HMI tags "2925RS001A01L02"
   "2925RS001A01L02.MSW" : 52809b66-421d-457f-8884-6f7a49d4e247 AT %DB5066.DBX18.0, 500 ms
   "2925RS001A01L02.DefaultText" : TextRef, internal   // Заголовок POPUP окна. При експорте из ECS через скрипт заполняется автоматически, если теги копируются в ручную то требуется в ручную задатать свойство Start Value
   "2925RS001A01L02.BlockInfo" : Array [0..2] of Int AT %DB5066.DBX38.0, 500 ms
   "2925RS001A01L02.StatusWork" : Int AT %DB5066.DBW242, 500 ms
   "2925RS001A01L02.FP_PARAM.DampingTime" : Int AT %DB5066.DBW50, 500 ms
   "2925RS001A01L02.FP_PARAM.Force_Value" : Real AT %DB5066.DBD52, 500 ms
   "2925RS001A01L02.FP_PARAM.Scale_Min" : Real AT %DB5066.DBD56, 500 ms
   "2925RS001A01L02.FP_PARAM.Scale_Max" : Real AT %DB5066.DBD60, 500 ms
   "2925RS001A01L02.FP_PARAM.Gradient" : Real AT %DB5066.DBD64, 500 ms
   "2925RS001A01L02.FP_PARAM.Grad_Pos" : Real AT %DB5066.DBD68, 500 ms
   "2925RS001A01L02.FP_PARAM.Grad_Neg" : Real AT %DB5066.DBD72, 500 ms
   "2925RS001A01L02.FP_PARAM.Grad_X" : Real AT %DB5066.DBD76, 500 ms
   "2925RS001A01L02.FP_PARAM.Gradient_Time_Pre" : Int AT %DB5066.DBW80, 500 ms
   "2925RS001A01L02.FP_PARAM.Gradient_Time_ACC" : Int AT %DB5066.DBW82, 500 ms
   "2925RS001A01L02.FP_PARAM.Alarm_Hyst" : Real AT %DB5066.DBD84, 500 ms
   "2925RS001A01L02.FP_PARAM.AlarmLimit_H3" : Real AT %DB5066.DBD88, 500 ms
   "2925RS001A01L02.FP_PARAM.AlarmLimit_H2" : Real AT %DB5066.DBD92, 500 ms
   "2925RS001A01L02.FP_PARAM.AlarmLimit_H1" : Real AT %DB5066.DBD96, 500 ms
   "2925RS001A01L02.FP_PARAM.AlarmLimit_L1" : Real AT %DB5066.DBD100, 500 ms
   "2925RS001A01L02.FP_PARAM.AlarmLimit_L2" : Real AT %DB5066.DBD104, 500 ms
   "2925RS001A01L02.FP_PARAM.AlarmLimit_L3" : Real AT %DB5066.DBD108, 500 ms
   "2925RS001A01L02.FP_PARAM.AlarmDelay_H3_Pre" : Int AT %DB5066.DBW112, 500 ms
   "2925RS001A01L02.FP_PARAM.AlarmDelay_H3_Acc" : Int AT %DB5066.DBW114, 500 ms
   "2925RS001A01L02.FP_PARAM.AlarmDelay_H2_Pre" : Int AT %DB5066.DBW116, 500 ms
   "2925RS001A01L02.FP_PARAM.AlarmDelay_H2_Acc" : Int AT %DB5066.DBW118, 500 ms
   "2925RS001A01L02.FP_PARAM.AlarmDelay_H1_Pre" : Int AT %DB5066.DBW120, 500 ms
   "2925RS001A01L02.FP_PARAM.AlarmDelay_H1_Acc" : Int AT %DB5066.DBW122, 500 ms
   "2925RS001A01L02.FP_PARAM.AlarmDelay_L1_Pre" : Int AT %DB5066.DBW124, 500 ms
   "2925RS001A01L02.FP_PARAM.AlarmDelay_L1_Acc" : Int AT %DB5066.DBW126, 500 ms
   "2925RS001A01L02.FP_PARAM.AlarmDelay_L2_Pre" : Int AT %DB5066.DBW128, 500 ms
   "2925RS001A01L02.FP_PARAM.AlarmDelay_L2_Acc" : Int AT %DB5066.DBW130, 500 ms
   "2925RS001A01L02.FP_PARAM.AlarmDelay_L3_Pre" : Int AT %DB5066.DBW132, 500 ms
   "2925RS001A01L02.FP_PARAM.AlarmDelay_L3_Acc" : Int AT %DB5066.DBW134, 500 ms
   "2925RS001A01L02.FP_PARAM.OpenLoopDelay_Pre" : Int AT %DB5066.DBW136, 500 ms
   "2925RS001A01L02.FP_PARAM.OpenLoopDelay_Acc" : Int AT %DB5066.DBW138, 500 ms
   "2925RS001A01L02.FP_PARAM.OverRangeDelay_Pre" : Int AT %DB5066.DBW140, 500 ms
   "2925RS001A01L02.FP_PARAM.OverRangeDelay_Acc" : Int AT %DB5066.DBW142, 500 ms
   "2925RS001A01L02.FP_PARAM.AuxLimit_H2_Value" : Real AT %DB5066.DBD144, 500 ms
   "2925RS001A01L02.FP_PARAM.AuxLimit_H1_Value" : Real AT %DB5066.DBD148, 500 ms
   "2925RS001A01L02.FP_PARAM.AuxLimit_L2_Value" : Real AT %DB5066.DBD152, 500 ms
   "2925RS001A01L02.FP_PARAM.AuxLimit_L1_Value" : Real AT %DB5066.DBD156, 500 ms
   "2925RS001A01L02.Unit" : TextRef, internal   // Еденицы измерения При експорте из ECS через скрипт заполняется автоматически, если теги копируются в ручную то требуется задатать свойство Text
   "2925RS001A01L02.Decimals" : TextRef, internal   // Формат отображения При експорте из ECS через скрипт, заполняется автоматически. Если теги копируются в ручную то требуется задатать свойство Text s999999.9
   "2925RS001A01L02.FP_EN.Square" : Bool AT %DB5066.DBX46.0, 500 ms
   "2925RS001A01L02.FP_EN.SquareRoot" : Bool AT %DB5066.DBX46.1, 500 ms
   "2925RS001A01L02.FP_EN.ParentSupress" : Bool AT %DB5066.DBX46.2, 500 ms
   "2925RS001A01L02.FP_EN.ParentSupressUnit" : Bool AT %DB5066.DBX46.3, 500 ms
   "2925RS001A01L02.FP_EN.Force" : Bool AT %DB5066.DBX46.4, 500 ms
   "2925RS001A01L02.FP_EN.Damping" : Bool AT %DB5066.DBX46.5, 500 ms
   "2925RS001A01L02.FP_EN.Gradient_Pos" : Bool AT %DB5066.DBX46.6, 500 ms
   "2925RS001A01L02.FP_EN.Gradient_Neg" : Bool AT %DB5066.DBX46.7, 500 ms
   "2925RS001A01L02.FP_EN.Hysteresis" : Bool AT %DB5066.DBX47.0, 500 ms
   "2925RS001A01L02.FP_EN.Alarm_H3" : Bool AT %DB5066.DBX47.1, 500 ms
   "2925RS001A01L02.FP_EN.Alarm_H2" : Bool AT %DB5066.DBX47.2, 500 ms
   "2925RS001A01L02.FP_EN.Alarm_H1" : Bool AT %DB5066.DBX47.3, 500 ms
   "2925RS001A01L02.FP_EN.Alarm_L1" : Bool AT %DB5066.DBX47.4, 500 ms
   "2925RS001A01L02.FP_EN.Alarm_L2" : Bool AT %DB5066.DBX47.5, 500 ms
   "2925RS001A01L02.FP_EN.Alarm_L3" : Bool AT %DB5066.DBX47.6, 500 ms
   "2925RS001A01L02.FP_EN.AlarmDelay_H3" : Bool AT %DB5066.DBX47.7, 500 ms
   "2925RS001A01L02.FP_EN.AlarmDelay_H2" : Bool AT %DB5066.DBX48.0, 500 ms
   "2925RS001A01L02.FP_EN.AlarmDelay_H1" : Bool AT %DB5066.DBX48.1, 500 ms
   "2925RS001A01L02.FP_EN.AlarmDelay_L1" : Bool AT %DB5066.DBX48.2, 500 ms
   "2925RS001A01L02.FP_EN.AlarmDelay_L2" : Bool AT %DB5066.DBX48.3, 500 ms
   "2925RS001A01L02.FP_EN.AlarmDelay_L3" : Bool AT %DB5066.DBX48.4, 500 ms
   "2925RS001A01L02.FP_EN.ROC_Warn" : Bool AT %DB5066.DBX48.5, 500 ms
   "2925RS001A01L02.FP_EN.U_Range_Warn" : Bool AT %DB5066.DBX48.6, 500 ms
   "2925RS001A01L02.FP_EN.O_Range_Warn" : Bool AT %DB5066.DBX48.7, 500 ms
   "2925RS001A01L02.trend_tag_name" : TextRef, internal   // Еденицы измерения При експорте из ECS через скрипт - заполняется автоматически, если теги копируются в ручную то требуется задатать свойство Text - имя тега для тренда
   "2925RS001A01L02.DQ.AL_H3" : Bool AT %DB5066.DBX16.0, 500 ms
   "2925RS001A01L02.DQ.AL_H2" : Bool AT %DB5066.DBX16.1, 500 ms
   "2925RS001A01L02.DQ.AL_H1" : Bool AT %DB5066.DBX16.2, 500 ms
   "2925RS001A01L02.DQ.AL_L1" : Bool AT %DB5066.DBX16.3, 500 ms
   "2925RS001A01L02.DQ.AL_L2" : Bool AT %DB5066.DBX16.4, 500 ms
   "2925RS001A01L02.DQ.AL_L3" : Bool AT %DB5066.DBX16.5, 500 ms
   "2925RS001A01L02.DQ.SIG_OK" : Bool AT %DB5066.DBX16.6, 500 ms
   "2925RS001A01L02.DQ.LIM_H2" : Bool AT %DB5066.DBX16.7, 500 ms
   "2925RS001A01L02.DQ.LIM_H1" : Bool AT %DB5066.DBX17.0, 500 ms
   "2925RS001A01L02.DQ.LIM_L1" : Bool AT %DB5066.DBX17.1, 500 ms
   "2925RS001A01L02.DQ.LIM_L2" : Bool AT %DB5066.DBX17.2, 500 ms
   "2925RS001A01L02.DQ.GR_P" : Bool AT %DB5066.DBX17.3, 500 ms
   "2925RS001A01L02.DQ.GR_N" : Bool AT %DB5066.DBX17.4, 500 ms
   "2925RS001A01L02.I.IN" : Real AT %DB5066.DBD2, 500 ms
   "2925RS001A01L02.I.SIG_TYPE" : Int AT %DB5066.DBW0, 500 ms
   "2925RS001A01L02.I.FI_BUS" : Byte AT %DB5066.DBB6, 500 ms
   "2925RS001A01L02.DI.U_RANGE" : Bool AT %DB5066.DBX7.0, 500 ms
   "2925RS001A01L02.DI.O_RANGE" : Bool AT %DB5066.DBX7.1, 500 ms
   "2925RS001A01L02.DI.SIG_FAULT" : Bool AT %DB5066.DBX7.2, 500 ms
   "2925RS001A01L02.DI.EnConfig" : Bool AT %DB5066.DBX7.3, 500 ms
   "2925RS001A01L02.DI.AEN" : Bool AT %DB5066.DBX7.4, 500 ms
   "2925RS001A01L02.DI.AL_SUPR" : Bool AT %DB5066.DBX7.5, 500 ms
   "2925RS001A01L02.Q.PV_NORM" : Real AT %DB5066.DBD8, 500 ms
   "2925RS001A01L02.Q.PV_SCAL" : Real AT %DB5066.DBD12, 500 ms
   "2925RS001A01L02.ParentInfo" : TextRef, internal   // Имя родителя для попап окна, вкладка инфо. При експорте из ECS через скрипт заполняется автоматически, если теги копируются в ручную то требуется в ручную задатать свойство Start Value

HMI tags "2925RS001A01T01"
   "2925RS001A01T01.MSW" : 52809b66-421d-457f-8884-6f7a49d4e247 AT %DB5067.DBX18.0, 500 ms
   "2925RS001A01T01.DefaultText" : TextRef, internal   // Заголовок POPUP окна. При експорте из ECS через скрипт заполняется автоматически, если теги копируются в ручную то требуется в ручную задатать свойство Start Value
   "2925RS001A01T01.BlockInfo" : Array [0..2] of Int AT %DB5067.DBX38.0, 500 ms
   "2925RS001A01T01.StatusWork" : Int AT %DB5067.DBW242, 500 ms
   "2925RS001A01T01.FP_PARAM.DampingTime" : Int AT %DB5067.DBW50, 500 ms
   "2925RS001A01T01.FP_PARAM.Force_Value" : Real AT %DB5067.DBD52, 500 ms
   "2925RS001A01T01.FP_PARAM.Scale_Min" : Real AT %DB5067.DBD56, 500 ms
   "2925RS001A01T01.FP_PARAM.Scale_Max" : Real AT %DB5067.DBD60, 500 ms
   "2925RS001A01T01.FP_PARAM.Gradient" : Real AT %DB5067.DBD64, 500 ms
   "2925RS001A01T01.FP_PARAM.Grad_Pos" : Real AT %DB5067.DBD68, 500 ms
   "2925RS001A01T01.FP_PARAM.Grad_Neg" : Real AT %DB5067.DBD72, 500 ms
   "2925RS001A01T01.FP_PARAM.Grad_X" : Real AT %DB5067.DBD76, 500 ms
   "2925RS001A01T01.FP_PARAM.Gradient_Time_Pre" : Int AT %DB5067.DBW80, 500 ms
   "2925RS001A01T01.FP_PARAM.Gradient_Time_ACC" : Int AT %DB5067.DBW82, 500 ms
   "2925RS001A01T01.FP_PARAM.Alarm_Hyst" : Real AT %DB5067.DBD84, 500 ms
   "2925RS001A01T01.FP_PARAM.AlarmLimit_H3" : Real AT %DB5067.DBD88, 500 ms
   "2925RS001A01T01.FP_PARAM.AlarmLimit_H2" : Real AT %DB5067.DBD92, 500 ms
   "2925RS001A01T01.FP_PARAM.AlarmLimit_H1" : Real AT %DB5067.DBD96, 500 ms
   "2925RS001A01T01.FP_PARAM.AlarmLimit_L1" : Real AT %DB5067.DBD100, 500 ms
   "2925RS001A01T01.FP_PARAM.AlarmLimit_L2" : Real AT %DB5067.DBD104, 500 ms
   "2925RS001A01T01.FP_PARAM.AlarmLimit_L3" : Real AT %DB5067.DBD108, 500 ms
   "2925RS001A01T01.FP_PARAM.AlarmDelay_H3_Pre" : Int AT %DB5067.DBW112, 500 ms
   "2925RS001A01T01.FP_PARAM.AlarmDelay_H3_Acc" : Int AT %DB5067.DBW114, 500 ms
   "2925RS001A01T01.FP_PARAM.AlarmDelay_H2_Pre" : Int AT %DB5067.DBW116, 500 ms
   "2925RS001A01T01.FP_PARAM.AlarmDelay_H2_Acc" : Int AT %DB5067.DBW118, 500 ms
   "2925RS001A01T01.FP_PARAM.AlarmDelay_H1_Pre" : Int AT %DB5067.DBW120, 500 ms
   "2925RS001A01T01.FP_PARAM.AlarmDelay_H1_Acc" : Int AT %DB5067.DBW122, 500 ms
   "2925RS001A01T01.FP_PARAM.AlarmDelay_L1_Pre" : Int AT %DB5067.DBW124, 500 ms
   "2925RS001A01T01.FP_PARAM.AlarmDelay_L1_Acc" : Int AT %DB5067.DBW126, 500 ms
   "2925RS001A01T01.FP_PARAM.AlarmDelay_L2_Pre" : Int AT %DB5067.DBW128, 500 ms
   "2925RS001A01T01.FP_PARAM.AlarmDelay_L2_Acc" : Int AT %DB5067.DBW130, 500 ms
   "2925RS001A01T01.FP_PARAM.AlarmDelay_L3_Pre" : Int AT %DB5067.DBW132, 500 ms
   "2925RS001A01T01.FP_PARAM.AlarmDelay_L3_Acc" : Int AT %DB5067.DBW134, 500 ms
   "2925RS001A01T01.FP_PARAM.OpenLoopDelay_Pre" : Int AT %DB5067.DBW136, 500 ms
   "2925RS001A01T01.FP_PARAM.OpenLoopDelay_Acc" : Int AT %DB5067.DBW138, 500 ms
   "2925RS001A01T01.FP_PARAM.OverRangeDelay_Pre" : Int AT %DB5067.DBW140, 500 ms
   "2925RS001A01T01.FP_PARAM.OverRangeDelay_Acc" : Int AT %DB5067.DBW142, 500 ms
   "2925RS001A01T01.FP_PARAM.AuxLimit_H2_Value" : Real AT %DB5067.DBD144, 500 ms
   "2925RS001A01T01.FP_PARAM.AuxLimit_H1_Value" : Real AT %DB5067.DBD148, 500 ms
   "2925RS001A01T01.FP_PARAM.AuxLimit_L2_Value" : Real AT %DB5067.DBD152, 500 ms
   "2925RS001A01T01.FP_PARAM.AuxLimit_L1_Value" : Real AT %DB5067.DBD156, 500 ms
   "2925RS001A01T01.Unit" : TextRef, internal   // Еденицы измерения При експорте из ECS через скрипт заполняется автоматически, если теги копируются в ручную то требуется задатать свойство Text
   "2925RS001A01T01.Decimals" : TextRef, internal   // Формат отображения При експорте из ECS через скрипт, заполняется автоматически. Если теги копируются в ручную то требуется задатать свойство Text s999999.9
   "2925RS001A01T01.FP_EN.Square" : Bool AT %DB5067.DBX46.0, 500 ms
   "2925RS001A01T01.FP_EN.SquareRoot" : Bool AT %DB5067.DBX46.1, 500 ms
   "2925RS001A01T01.FP_EN.ParentSupress" : Bool AT %DB5067.DBX46.2, 500 ms
   "2925RS001A01T01.FP_EN.ParentSupressUnit" : Bool AT %DB5067.DBX46.3, 500 ms
   "2925RS001A01T01.FP_EN.Force" : Bool AT %DB5067.DBX46.4, 500 ms
   "2925RS001A01T01.FP_EN.Damping" : Bool AT %DB5067.DBX46.5, 500 ms
   "2925RS001A01T01.FP_EN.Gradient_Pos" : Bool AT %DB5067.DBX46.6, 500 ms
   "2925RS001A01T01.FP_EN.Gradient_Neg" : Bool AT %DB5067.DBX46.7, 500 ms
   "2925RS001A01T01.FP_EN.Hysteresis" : Bool AT %DB5067.DBX47.0, 500 ms
   "2925RS001A01T01.FP_EN.Alarm_H3" : Bool AT %DB5067.DBX47.1, 500 ms
   "2925RS001A01T01.FP_EN.Alarm_H2" : Bool AT %DB5067.DBX47.2, 500 ms
   "2925RS001A01T01.FP_EN.Alarm_H1" : Bool AT %DB5067.DBX47.3, 500 ms
   "2925RS001A01T01.FP_EN.Alarm_L1" : Bool AT %DB5067.DBX47.4, 500 ms
   "2925RS001A01T01.FP_EN.Alarm_L2" : Bool AT %DB5067.DBX47.5, 500 ms
   "2925RS001A01T01.FP_EN.Alarm_L3" : Bool AT %DB5067.DBX47.6, 500 ms
   "2925RS001A01T01.FP_EN.AlarmDelay_H3" : Bool AT %DB5067.DBX47.7, 500 ms
   "2925RS001A01T01.FP_EN.AlarmDelay_H2" : Bool AT %DB5067.DBX48.0, 500 ms
   "2925RS001A01T01.FP_EN.AlarmDelay_H1" : Bool AT %DB5067.DBX48.1, 500 ms
   "2925RS001A01T01.FP_EN.AlarmDelay_L1" : Bool AT %DB5067.DBX48.2, 500 ms
   "2925RS001A01T01.FP_EN.AlarmDelay_L2" : Bool AT %DB5067.DBX48.3, 500 ms
   "2925RS001A01T01.FP_EN.AlarmDelay_L3" : Bool AT %DB5067.DBX48.4, 500 ms
   "2925RS001A01T01.FP_EN.ROC_Warn" : Bool AT %DB5067.DBX48.5, 500 ms
   "2925RS001A01T01.FP_EN.U_Range_Warn" : Bool AT %DB5067.DBX48.6, 500 ms
   "2925RS001A01T01.FP_EN.O_Range_Warn" : Bool AT %DB5067.DBX48.7, 500 ms
   "2925RS001A01T01.trend_tag_name" : TextRef, internal   // Еденицы измерения При експорте из ECS через скрипт - заполняется автоматически, если теги копируются в ручную то требуется задатать свойство Text - имя тега для тренда
   "2925RS001A01T01.DQ.AL_H3" : Bool AT %DB5067.DBX16.0, 500 ms
   "2925RS001A01T01.DQ.AL_H2" : Bool AT %DB5067.DBX16.1, 500 ms
   "2925RS001A01T01.DQ.AL_H1" : Bool AT %DB5067.DBX16.2, 500 ms
   "2925RS001A01T01.DQ.AL_L1" : Bool AT %DB5067.DBX16.3, 500 ms
   "2925RS001A01T01.DQ.AL_L2" : Bool AT %DB5067.DBX16.4, 500 ms
   "2925RS001A01T01.DQ.AL_L3" : Bool AT %DB5067.DBX16.5, 500 ms
   "2925RS001A01T01.DQ.SIG_OK" : Bool AT %DB5067.DBX16.6, 500 ms
   "2925RS001A01T01.DQ.LIM_H2" : Bool AT %DB5067.DBX16.7, 500 ms
   "2925RS001A01T01.DQ.LIM_H1" : Bool AT %DB5067.DBX17.0, 500 ms
   "2925RS001A01T01.DQ.LIM_L1" : Bool AT %DB5067.DBX17.1, 500 ms
   "2925RS001A01T01.DQ.LIM_L2" : Bool AT %DB5067.DBX17.2, 500 ms
   "2925RS001A01T01.DQ.GR_P" : Bool AT %DB5067.DBX17.3, 500 ms
   "2925RS001A01T01.DQ.GR_N" : Bool AT %DB5067.DBX17.4, 500 ms
   "2925RS001A01T01.I.IN" : Real AT %DB5067.DBD2, 500 ms
   "2925RS001A01T01.I.SIG_TYPE" : Int AT %DB5067.DBW0, 500 ms
   "2925RS001A01T01.I.FI_BUS" : Byte AT %DB5067.DBB6, 500 ms
   "2925RS001A01T01.DI.U_RANGE" : Bool AT %DB5067.DBX7.0, 500 ms
   "2925RS001A01T01.DI.O_RANGE" : Bool AT %DB5067.DBX7.1, 500 ms
   "2925RS001A01T01.DI.SIG_FAULT" : Bool AT %DB5067.DBX7.2, 500 ms
   "2925RS001A01T01.DI.EnConfig" : Bool AT %DB5067.DBX7.3, 500 ms
   "2925RS001A01T01.DI.AEN" : Bool AT %DB5067.DBX7.4, 500 ms
   "2925RS001A01T01.DI.AL_SUPR" : Bool AT %DB5067.DBX7.5, 500 ms
   "2925RS001A01T01.Q.PV_NORM" : Real AT %DB5067.DBD8, 500 ms
   "2925RS001A01T01.Q.PV_SCAL" : Real AT %DB5067.DBD12, 500 ms
   "2925RS001A01T01.ParentInfo" : TextRef, internal   // Имя родителя для попап окна, вкладка инфо. При експорте из ECS через скрипт заполняется автоматически, если теги копируются в ручную то требуется в ручную задатать свойство Start Value

HMI tags "2925RS001A01T02"
   "2925RS001A01T02.MSW" : 52809b66-421d-457f-8884-6f7a49d4e247 AT %DB5068.DBX18.0, 500 ms
   "2925RS001A01T02.DefaultText" : TextRef, internal   // Заголовок POPUP окна. При експорте из ECS через скрипт заполняется автоматически, если теги копируются в ручную то требуется в ручную задатать свойство Start Value
   "2925RS001A01T02.BlockInfo" : Array [0..2] of Int AT %DB5068.DBX38.0, 500 ms
   "2925RS001A01T02.StatusWork" : Int AT %DB5068.DBW242, 500 ms
   "2925RS001A01T02.FP_PARAM.DampingTime" : Int AT %DB5068.DBW50, 500 ms
   "2925RS001A01T02.FP_PARAM.Force_Value" : Real AT %DB5068.DBD52, 500 ms
   "2925RS001A01T02.FP_PARAM.Scale_Min" : Real AT %DB5068.DBD56, 500 ms
   "2925RS001A01T02.FP_PARAM.Scale_Max" : Real AT %DB5068.DBD60, 500 ms
   "2925RS001A01T02.FP_PARAM.Gradient" : Real AT %DB5068.DBD64, 500 ms
   "2925RS001A01T02.FP_PARAM.Grad_Pos" : Real AT %DB5068.DBD68, 500 ms
   "2925RS001A01T02.FP_PARAM.Grad_Neg" : Real AT %DB5068.DBD72, 500 ms
   "2925RS001A01T02.FP_PARAM.Grad_X" : Real AT %DB5068.DBD76, 500 ms
   "2925RS001A01T02.FP_PARAM.Gradient_Time_Pre" : Int AT %DB5068.DBW80, 500 ms
   "2925RS001A01T02.FP_PARAM.Gradient_Time_ACC" : Int AT %DB5068.DBW82, 500 ms
   "2925RS001A01T02.FP_PARAM.Alarm_Hyst" : Real AT %DB5068.DBD84, 500 ms
   "2925RS001A01T02.FP_PARAM.AlarmLimit_H3" : Real AT %DB5068.DBD88, 500 ms
   "2925RS001A01T02.FP_PARAM.AlarmLimit_H2" : Real AT %DB5068.DBD92, 500 ms
   "2925RS001A01T02.FP_PARAM.AlarmLimit_H1" : Real AT %DB5068.DBD96, 500 ms
   "2925RS001A01T02.FP_PARAM.AlarmLimit_L1" : Real AT %DB5068.DBD100, 500 ms
   "2925RS001A01T02.FP_PARAM.AlarmLimit_L2" : Real AT %DB5068.DBD104, 500 ms
   "2925RS001A01T02.FP_PARAM.AlarmLimit_L3" : Real AT %DB5068.DBD108, 500 ms
   "2925RS001A01T02.FP_PARAM.AlarmDelay_H3_Pre" : Int AT %DB5068.DBW112, 500 ms
   "2925RS001A01T02.FP_PARAM.AlarmDelay_H3_Acc" : Int AT %DB5068.DBW114, 500 ms
   "2925RS001A01T02.FP_PARAM.AlarmDelay_H2_Pre" : Int AT %DB5068.DBW116, 500 ms
   "2925RS001A01T02.FP_PARAM.AlarmDelay_H2_Acc" : Int AT %DB5068.DBW118, 500 ms
   "2925RS001A01T02.FP_PARAM.AlarmDelay_H1_Pre" : Int AT %DB5068.DBW120, 500 ms
   "2925RS001A01T02.FP_PARAM.AlarmDelay_H1_Acc" : Int AT %DB5068.DBW122, 500 ms
   "2925RS001A01T02.FP_PARAM.AlarmDelay_L1_Pre" : Int AT %DB5068.DBW124, 500 ms
   "2925RS001A01T02.FP_PARAM.AlarmDelay_L1_Acc" : Int AT %DB5068.DBW126, 500 ms
   "2925RS001A01T02.FP_PARAM.AlarmDelay_L2_Pre" : Int AT %DB5068.DBW128, 500 ms
   "2925RS001A01T02.FP_PARAM.AlarmDelay_L2_Acc" : Int AT %DB5068.DBW130, 500 ms
   "2925RS001A01T02.FP_PARAM.AlarmDelay_L3_Pre" : Int AT %DB5068.DBW132, 500 ms
   "2925RS001A01T02.FP_PARAM.AlarmDelay_L3_Acc" : Int AT %DB5068.DBW134, 500 ms
   "2925RS001A01T02.FP_PARAM.OpenLoopDelay_Pre" : Int AT %DB5068.DBW136, 500 ms
   "2925RS001A01T02.FP_PARAM.OpenLoopDelay_Acc" : Int AT %DB5068.DBW138, 500 ms
   "2925RS001A01T02.FP_PARAM.OverRangeDelay_Pre" : Int AT %DB5068.DBW140, 500 ms
   "2925RS001A01T02.FP_PARAM.OverRangeDelay_Acc" : Int AT %DB5068.DBW142, 500 ms
   "2925RS001A01T02.FP_PARAM.AuxLimit_H2_Value" : Real AT %DB5068.DBD144, 500 ms
   "2925RS001A01T02.FP_PARAM.AuxLimit_H1_Value" : Real AT %DB5068.DBD148, 500 ms
   "2925RS001A01T02.FP_PARAM.AuxLimit_L2_Value" : Real AT %DB5068.DBD152, 500 ms
   "2925RS001A01T02.FP_PARAM.AuxLimit_L1_Value" : Real AT %DB5068.DBD156, 500 ms
   "2925RS001A01T02.Unit" : TextRef, internal   // Еденицы измерения При експорте из ECS через скрипт заполняется автоматически, если теги копируются в ручную то требуется задатать свойство Text
   "2925RS001A01T02.Decimals" : TextRef, internal   // Формат отображения При експорте из ECS через скрипт, заполняется автоматически. Если теги копируются в ручную то требуется задатать свойство Text s999999.9
   "2925RS001A01T02.FP_EN.Square" : Bool AT %DB5068.DBX46.0, 500 ms
   "2925RS001A01T02.FP_EN.SquareRoot" : Bool AT %DB5068.DBX46.1, 500 ms
   "2925RS001A01T02.FP_EN.ParentSupress" : Bool AT %DB5068.DBX46.2, 500 ms
   "2925RS001A01T02.FP_EN.ParentSupressUnit" : Bool AT %DB5068.DBX46.3, 500 ms
   "2925RS001A01T02.FP_EN.Force" : Bool AT %DB5068.DBX46.4, 500 ms
   "2925RS001A01T02.FP_EN.Damping" : Bool AT %DB5068.DBX46.5, 500 ms
   "2925RS001A01T02.FP_EN.Gradient_Pos" : Bool AT %DB5068.DBX46.6, 500 ms
   "2925RS001A01T02.FP_EN.Gradient_Neg" : Bool AT %DB5068.DBX46.7, 500 ms
   "2925RS001A01T02.FP_EN.Hysteresis" : Bool AT %DB5068.DBX47.0, 500 ms
   "2925RS001A01T02.FP_EN.Alarm_H3" : Bool AT %DB5068.DBX47.1, 500 ms
   "2925RS001A01T02.FP_EN.Alarm_H2" : Bool AT %DB5068.DBX47.2, 500 ms
   "2925RS001A01T02.FP_EN.Alarm_H1" : Bool AT %DB5068.DBX47.3, 500 ms
   "2925RS001A01T02.FP_EN.Alarm_L1" : Bool AT %DB5068.DBX47.4, 500 ms
   "2925RS001A01T02.FP_EN.Alarm_L2" : Bool AT %DB5068.DBX47.5, 500 ms
   "2925RS001A01T02.FP_EN.Alarm_L3" : Bool AT %DB5068.DBX47.6, 500 ms
   "2925RS001A01T02.FP_EN.AlarmDelay_H3" : Bool AT %DB5068.DBX47.7, 500 ms
   "2925RS001A01T02.FP_EN.AlarmDelay_H2" : Bool AT %DB5068.DBX48.0, 500 ms
   "2925RS001A01T02.FP_EN.AlarmDelay_H1" : Bool AT %DB5068.DBX48.1, 500 ms
   "2925RS001A01T02.FP_EN.AlarmDelay_L1" : Bool AT %DB5068.DBX48.2, 500 ms
   "2925RS001A01T02.FP_EN.AlarmDelay_L2" : Bool AT %DB5068.DBX48.3, 500 ms
   "2925RS001A01T02.FP_EN.AlarmDelay_L3" : Bool AT %DB5068.DBX48.4, 500 ms
   "2925RS001A01T02.FP_EN.ROC_Warn" : Bool AT %DB5068.DBX48.5, 500 ms
   "2925RS001A01T02.FP_EN.U_Range_Warn" : Bool AT %DB5068.DBX48.6, 500 ms
   "2925RS001A01T02.FP_EN.O_Range_Warn" : Bool AT %DB5068.DBX48.7, 500 ms
   "2925RS001A01T02.trend_tag_name" : TextRef, internal   // Еденицы измерения При експорте из ECS через скрипт - заполняется автоматически, если теги копируются в ручную то требуется задатать свойство Text - имя тега для тренда
   "2925RS001A01T02.DQ.AL_H3" : Bool AT %DB5068.DBX16.0, 500 ms
   "2925RS001A01T02.DQ.AL_H2" : Bool AT %DB5068.DBX16.1, 500 ms
   "2925RS001A01T02.DQ.AL_H1" : Bool AT %DB5068.DBX16.2, 500 ms
   "2925RS001A01T02.DQ.AL_L1" : Bool AT %DB5068.DBX16.3, 500 ms
   "2925RS001A01T02.DQ.AL_L2" : Bool AT %DB5068.DBX16.4, 500 ms
   "2925RS001A01T02.DQ.AL_L3" : Bool AT %DB5068.DBX16.5, 500 ms
   "2925RS001A01T02.DQ.SIG_OK" : Bool AT %DB5068.DBX16.6, 500 ms
   "2925RS001A01T02.DQ.LIM_H2" : Bool AT %DB5068.DBX16.7, 500 ms
   "2925RS001A01T02.DQ.LIM_H1" : Bool AT %DB5068.DBX17.0, 500 ms
   "2925RS001A01T02.DQ.LIM_L1" : Bool AT %DB5068.DBX17.1, 500 ms
   "2925RS001A01T02.DQ.LIM_L2" : Bool AT %DB5068.DBX17.2, 500 ms
   "2925RS001A01T02.DQ.GR_P" : Bool AT %DB5068.DBX17.3, 500 ms
   "2925RS001A01T02.DQ.GR_N" : Bool AT %DB5068.DBX17.4, 500 ms
   "2925RS001A01T02.I.IN" : Real AT %DB5068.DBD2, 500 ms
   "2925RS001A01T02.I.SIG_TYPE" : Int AT %DB5068.DBW0, 500 ms
   "2925RS001A01T02.I.FI_BUS" : Byte AT %DB5068.DBB6, 500 ms
   "2925RS001A01T02.DI.U_RANGE" : Bool AT %DB5068.DBX7.0, 500 ms
   "2925RS001A01T02.DI.O_RANGE" : Bool AT %DB5068.DBX7.1, 500 ms
   "2925RS001A01T02.DI.SIG_FAULT" : Bool AT %DB5068.DBX7.2, 500 ms
   "2925RS001A01T02.DI.EnConfig" : Bool AT %DB5068.DBX7.3, 500 ms
   "2925RS001A01T02.DI.AEN" : Bool AT %DB5068.DBX7.4, 500 ms
   "2925RS001A01T02.DI.AL_SUPR" : Bool AT %DB5068.DBX7.5, 500 ms
   "2925RS001A01T02.Q.PV_NORM" : Real AT %DB5068.DBD8, 500 ms
   "2925RS001A01T02.Q.PV_SCAL" : Real AT %DB5068.DBD12, 500 ms
   "2925RS001A01T02.ParentInfo" : TextRef, internal   // Имя родителя для попап окна, вкладка инфо. При експорте из ECS через скрипт заполняется автоматически, если теги копируются в ручную то требуется в ручную задатать свойство Start Value

HMI tags "2925RS001A01T03"
   "2925RS001A01T03.MSW" : 52809b66-421d-457f-8884-6f7a49d4e247 AT %DB5069.DBX18.0, 500 ms
   "2925RS001A01T03.DefaultText" : TextRef, internal   // Заголовок POPUP окна. При експорте из ECS через скрипт заполняется автоматически, если теги копируются в ручную то требуется в ручную задатать свойство Start Value
   "2925RS001A01T03.BlockInfo" : Array [0..2] of Int AT %DB5069.DBX38.0, 500 ms
   "2925RS001A01T03.StatusWork" : Int AT %DB5069.DBW242, 500 ms
   "2925RS001A01T03.FP_PARAM.DampingTime" : Int AT %DB5069.DBW50, 500 ms
   "2925RS001A01T03.FP_PARAM.Force_Value" : Real AT %DB5069.DBD52, 500 ms
   "2925RS001A01T03.FP_PARAM.Scale_Min" : Real AT %DB5069.DBD56, 500 ms
   "2925RS001A01T03.FP_PARAM.Scale_Max" : Real AT %DB5069.DBD60, 500 ms
   "2925RS001A01T03.FP_PARAM.Gradient" : Real AT %DB5069.DBD64, 500 ms
   "2925RS001A01T03.FP_PARAM.Grad_Pos" : Real AT %DB5069.DBD68, 500 ms
   "2925RS001A01T03.FP_PARAM.Grad_Neg" : Real AT %DB5069.DBD72, 500 ms
   "2925RS001A01T03.FP_PARAM.Grad_X" : Real AT %DB5069.DBD76, 500 ms
   "2925RS001A01T03.FP_PARAM.Gradient_Time_Pre" : Int AT %DB5069.DBW80, 500 ms
   "2925RS001A01T03.FP_PARAM.Gradient_Time_ACC" : Int AT %DB5069.DBW82, 500 ms
   "2925RS001A01T03.FP_PARAM.Alarm_Hyst" : Real AT %DB5069.DBD84, 500 ms
   "2925RS001A01T03.FP_PARAM.AlarmLimit_H3" : Real AT %DB5069.DBD88, 500 ms
   "2925RS001A01T03.FP_PARAM.AlarmLimit_H2" : Real AT %DB5069.DBD92, 500 ms
   "2925RS001A01T03.FP_PARAM.AlarmLimit_H1" : Real AT %DB5069.DBD96, 500 ms
   "2925RS001A01T03.FP_PARAM.AlarmLimit_L1" : Real AT %DB5069.DBD100, 500 ms
   "2925RS001A01T03.FP_PARAM.AlarmLimit_L2" : Real AT %DB5069.DBD104, 500 ms
   "2925RS001A01T03.FP_PARAM.AlarmLimit_L3" : Real AT %DB5069.DBD108, 500 ms
   "2925RS001A01T03.FP_PARAM.AlarmDelay_H3_Pre" : Int AT %DB5069.DBW112, 500 ms
   "2925RS001A01T03.FP_PARAM.AlarmDelay_H3_Acc" : Int AT %DB5069.DBW114, 500 ms
   "2925RS001A01T03.FP_PARAM.AlarmDelay_H2_Pre" : Int AT %DB5069.DBW116, 500 ms
   "2925RS001A01T03.FP_PARAM.AlarmDelay_H2_Acc" : Int AT %DB5069.DBW118, 500 ms
   "2925RS001A01T03.FP_PARAM.AlarmDelay_H1_Pre" : Int AT %DB5069.DBW120, 500 ms
   "2925RS001A01T03.FP_PARAM.AlarmDelay_H1_Acc" : Int AT %DB5069.DBW122, 500 ms
   "2925RS001A01T03.FP_PARAM.AlarmDelay_L1_Pre" : Int AT %DB5069.DBW124, 500 ms
   "2925RS001A01T03.FP_PARAM.AlarmDelay_L1_Acc" : Int AT %DB5069.DBW126, 500 ms
   "2925RS001A01T03.FP_PARAM.AlarmDelay_L2_Pre" : Int AT %DB5069.DBW128, 500 ms
   "2925RS001A01T03.FP_PARAM.AlarmDelay_L2_Acc" : Int AT %DB5069.DBW130, 500 ms
   "2925RS001A01T03.FP_PARAM.AlarmDelay_L3_Pre" : Int AT %DB5069.DBW132, 500 ms
   "2925RS001A01T03.FP_PARAM.AlarmDelay_L3_Acc" : Int AT %DB5069.DBW134, 500 ms
   "2925RS001A01T03.FP_PARAM.OpenLoopDelay_Pre" : Int AT %DB5069.DBW136, 500 ms
   "2925RS001A01T03.FP_PARAM.OpenLoopDelay_Acc" : Int AT %DB5069.DBW138, 500 ms
   "2925RS001A01T03.FP_PARAM.OverRangeDelay_Pre" : Int AT %DB5069.DBW140, 500 ms
   "2925RS001A01T03.FP_PARAM.OverRangeDelay_Acc" : Int AT %DB5069.DBW142, 500 ms
   "2925RS001A01T03.FP_PARAM.AuxLimit_H2_Value" : Real AT %DB5069.DBD144, 500 ms
   "2925RS001A01T03.FP_PARAM.AuxLimit_H1_Value" : Real AT %DB5069.DBD148, 500 ms
   "2925RS001A01T03.FP_PARAM.AuxLimit_L2_Value" : Real AT %DB5069.DBD152, 500 ms
   "2925RS001A01T03.FP_PARAM.AuxLimit_L1_Value" : Real AT %DB5069.DBD156, 500 ms
   "2925RS001A01T03.Unit" : TextRef, internal   // Еденицы измерения При експорте из ECS через скрипт заполняется автоматически, если теги копируются в ручную то требуется задатать свойство Text
   "2925RS001A01T03.Decimals" : TextRef, internal   // Формат отображения При експорте из ECS через скрипт, заполняется автоматически. Если теги копируются в ручную то требуется задатать свойство Text s999999.9
   "2925RS001A01T03.FP_EN.Square" : Bool AT %DB5069.DBX46.0, 500 ms
   "2925RS001A01T03.FP_EN.SquareRoot" : Bool AT %DB5069.DBX46.1, 500 ms
   "2925RS001A01T03.FP_EN.ParentSupress" : Bool AT %DB5069.DBX46.2, 500 ms
   "2925RS001A01T03.FP_EN.ParentSupressUnit" : Bool AT %DB5069.DBX46.3, 500 ms
   "2925RS001A01T03.FP_EN.Force" : Bool AT %DB5069.DBX46.4, 500 ms
   "2925RS001A01T03.FP_EN.Damping" : Bool AT %DB5069.DBX46.5, 500 ms
   "2925RS001A01T03.FP_EN.Gradient_Pos" : Bool AT %DB5069.DBX46.6, 500 ms
   "2925RS001A01T03.FP_EN.Gradient_Neg" : Bool AT %DB5069.DBX46.7, 500 ms
   "2925RS001A01T03.FP_EN.Hysteresis" : Bool AT %DB5069.DBX47.0, 500 ms
   "2925RS001A01T03.FP_EN.Alarm_H3" : Bool AT %DB5069.DBX47.1, 500 ms
   "2925RS001A01T03.FP_EN.Alarm_H2" : Bool AT %DB5069.DBX47.2, 500 ms
   "2925RS001A01T03.FP_EN.Alarm_H1" : Bool AT %DB5069.DBX47.3, 500 ms
   "2925RS001A01T03.FP_EN.Alarm_L1" : Bool AT %DB5069.DBX47.4, 500 ms
   "2925RS001A01T03.FP_EN.Alarm_L2" : Bool AT %DB5069.DBX47.5, 500 ms
   "2925RS001A01T03.FP_EN.Alarm_L3" : Bool AT %DB5069.DBX47.6, 500 ms
   "2925RS001A01T03.FP_EN.AlarmDelay_H3" : Bool AT %DB5069.DBX47.7, 500 ms
   "2925RS001A01T03.FP_EN.AlarmDelay_H2" : Bool AT %DB5069.DBX48.0, 500 ms
   "2925RS001A01T03.FP_EN.AlarmDelay_H1" : Bool AT %DB5069.DBX48.1, 500 ms
   "2925RS001A01T03.FP_EN.AlarmDelay_L1" : Bool AT %DB5069.DBX48.2, 500 ms
   "2925RS001A01T03.FP_EN.AlarmDelay_L2" : Bool AT %DB5069.DBX48.3, 500 ms
   "2925RS001A01T03.FP_EN.AlarmDelay_L3" : Bool AT %DB5069.DBX48.4, 500 ms
   "2925RS001A01T03.FP_EN.ROC_Warn" : Bool AT %DB5069.DBX48.5, 500 ms
   "2925RS001A01T03.FP_EN.U_Range_Warn" : Bool AT %DB5069.DBX48.6, 500 ms
   "2925RS001A01T03.FP_EN.O_Range_Warn" : Bool AT %DB5069.DBX48.7, 500 ms
   "2925RS001A01T03.trend_tag_name" : TextRef, internal   // Еденицы измерения При експорте из ECS через скрипт - заполняется автоматически, если теги копируются в ручную то требуется задатать свойство Text - имя тега для тренда
   "2925RS001A01T03.DQ.AL_H3" : Bool AT %DB5069.DBX16.0, 500 ms
   "2925RS001A01T03.DQ.AL_H2" : Bool AT %DB5069.DBX16.1, 500 ms
   "2925RS001A01T03.DQ.AL_H1" : Bool AT %DB5069.DBX16.2, 500 ms
   "2925RS001A01T03.DQ.AL_L1" : Bool AT %DB5069.DBX16.3, 500 ms
   "2925RS001A01T03.DQ.AL_L2" : Bool AT %DB5069.DBX16.4, 500 ms
   "2925RS001A01T03.DQ.AL_L3" : Bool AT %DB5069.DBX16.5, 500 ms
   "2925RS001A01T03.DQ.SIG_OK" : Bool AT %DB5069.DBX16.6, 500 ms
   "2925RS001A01T03.DQ.LIM_H2" : Bool AT %DB5069.DBX16.7, 500 ms
   "2925RS001A01T03.DQ.LIM_H1" : Bool AT %DB5069.DBX17.0, 500 ms
   "2925RS001A01T03.DQ.LIM_L1" : Bool AT %DB5069.DBX17.1, 500 ms
   "2925RS001A01T03.DQ.LIM_L2" : Bool AT %DB5069.DBX17.2, 500 ms
   "2925RS001A01T03.DQ.GR_P" : Bool AT %DB5069.DBX17.3, 500 ms
   "2925RS001A01T03.DQ.GR_N" : Bool AT %DB5069.DBX17.4, 500 ms
   "2925RS001A01T03.I.IN" : Real AT %DB5069.DBD2, 500 ms
   "2925RS001A01T03.I.SIG_TYPE" : Int AT %DB5069.DBW0, 500 ms
   "2925RS001A01T03.I.FI_BUS" : Byte AT %DB5069.DBB6, 500 ms
   "2925RS001A01T03.DI.U_RANGE" : Bool AT %DB5069.DBX7.0, 500 ms
   "2925RS001A01T03.DI.O_RANGE" : Bool AT %DB5069.DBX7.1, 500 ms
   "2925RS001A01T03.DI.SIG_FAULT" : Bool AT %DB5069.DBX7.2, 500 ms
   "2925RS001A01T03.DI.EnConfig" : Bool AT %DB5069.DBX7.3, 500 ms
   "2925RS001A01T03.DI.AEN" : Bool AT %DB5069.DBX7.4, 500 ms
   "2925RS001A01T03.DI.AL_SUPR" : Bool AT %DB5069.DBX7.5, 500 ms
   "2925RS001A01T03.Q.PV_NORM" : Real AT %DB5069.DBD8, 500 ms
   "2925RS001A01T03.Q.PV_SCAL" : Real AT %DB5069.DBD12, 500 ms
   "2925RS001A01T03.ParentInfo" : TextRef, internal   // Имя родителя для попап окна, вкладка инфо. При експорте из ECS через скрипт заполняется автоматически, если теги копируются в ручную то требуется в ручную задатать свойство Start Value

HMI tags "2925RS001A01T04"
   "2925RS001A01T04.MSW" : 52809b66-421d-457f-8884-6f7a49d4e247 AT %DB5070.DBX18.0, 500 ms
   "2925RS001A01T04.DefaultText" : TextRef, internal   // Заголовок POPUP окна. При експорте из ECS через скрипт заполняется автоматически, если теги копируются в ручную то требуется в ручную задатать свойство Start Value
   "2925RS001A01T04.BlockInfo" : Array [0..2] of Int AT %DB5070.DBX38.0, 500 ms
   "2925RS001A01T04.StatusWork" : Int AT %DB5070.DBW242, 500 ms
   "2925RS001A01T04.FP_PARAM.DampingTime" : Int AT %DB5070.DBW50, 500 ms
   "2925RS001A01T04.FP_PARAM.Force_Value" : Real AT %DB5070.DBD52, 500 ms
   "2925RS001A01T04.FP_PARAM.Scale_Min" : Real AT %DB5070.DBD56, 500 ms
   "2925RS001A01T04.FP_PARAM.Scale_Max" : Real AT %DB5070.DBD60, 500 ms
   "2925RS001A01T04.FP_PARAM.Gradient" : Real AT %DB5070.DBD64, 500 ms
   "2925RS001A01T04.FP_PARAM.Grad_Pos" : Real AT %DB5070.DBD68, 500 ms
   "2925RS001A01T04.FP_PARAM.Grad_Neg" : Real AT %DB5070.DBD72, 500 ms
   "2925RS001A01T04.FP_PARAM.Grad_X" : Real AT %DB5070.DBD76, 500 ms
   "2925RS001A01T04.FP_PARAM.Gradient_Time_Pre" : Int AT %DB5070.DBW80, 500 ms
   "2925RS001A01T04.FP_PARAM.Gradient_Time_ACC" : Int AT %DB5070.DBW82, 500 ms
   "2925RS001A01T04.FP_PARAM.Alarm_Hyst" : Real AT %DB5070.DBD84, 500 ms
   "2925RS001A01T04.FP_PARAM.AlarmLimit_H3" : Real AT %DB5070.DBD88, 500 ms
   "2925RS001A01T04.FP_PARAM.AlarmLimit_H2" : Real AT %DB5070.DBD92, 500 ms
   "2925RS001A01T04.FP_PARAM.AlarmLimit_H1" : Real AT %DB5070.DBD96, 500 ms
   "2925RS001A01T04.FP_PARAM.AlarmLimit_L1" : Real AT %DB5070.DBD100, 500 ms
   "2925RS001A01T04.FP_PARAM.AlarmLimit_L2" : Real AT %DB5070.DBD104, 500 ms
   "2925RS001A01T04.FP_PARAM.AlarmLimit_L3" : Real AT %DB5070.DBD108, 500 ms
   "2925RS001A01T04.FP_PARAM.AlarmDelay_H3_Pre" : Int AT %DB5070.DBW112, 500 ms
   "2925RS001A01T04.FP_PARAM.AlarmDelay_H3_Acc" : Int AT %DB5070.DBW114, 500 ms
   "2925RS001A01T04.FP_PARAM.AlarmDelay_H2_Pre" : Int AT %DB5070.DBW116, 500 ms
   "2925RS001A01T04.FP_PARAM.AlarmDelay_H2_Acc" : Int AT %DB5070.DBW118, 500 ms
   "2925RS001A01T04.FP_PARAM.AlarmDelay_H1_Pre" : Int AT %DB5070.DBW120, 500 ms
   "2925RS001A01T04.FP_PARAM.AlarmDelay_H1_Acc" : Int AT %DB5070.DBW122, 500 ms
   "2925RS001A01T04.FP_PARAM.AlarmDelay_L1_Pre" : Int AT %DB5070.DBW124, 500 ms
   "2925RS001A01T04.FP_PARAM.AlarmDelay_L1_Acc" : Int AT %DB5070.DBW126, 500 ms
   "2925RS001A01T04.FP_PARAM.AlarmDelay_L2_Pre" : Int AT %DB5070.DBW128, 500 ms
   "2925RS001A01T04.FP_PARAM.AlarmDelay_L2_Acc" : Int AT %DB5070.DBW130, 500 ms
   "2925RS001A01T04.FP_PARAM.AlarmDelay_L3_Pre" : Int AT %DB5070.DBW132, 500 ms
   "2925RS001A01T04.FP_PARAM.AlarmDelay_L3_Acc" : Int AT %DB5070.DBW134, 500 ms
   "2925RS001A01T04.FP_PARAM.OpenLoopDelay_Pre" : Int AT %DB5070.DBW136, 500 ms
   "2925RS001A01T04.FP_PARAM.OpenLoopDelay_Acc" : Int AT %DB5070.DBW138, 500 ms
   "2925RS001A01T04.FP_PARAM.OverRangeDelay_Pre" : Int AT %DB5070.DBW140, 500 ms
   "2925RS001A01T04.FP_PARAM.OverRangeDelay_Acc" : Int AT %DB5070.DBW142, 500 ms
   "2925RS001A01T04.FP_PARAM.AuxLimit_H2_Value" : Real AT %DB5070.DBD144, 500 ms
   "2925RS001A01T04.FP_PARAM.AuxLimit_H1_Value" : Real AT %DB5070.DBD148, 500 ms
   "2925RS001A01T04.FP_PARAM.AuxLimit_L2_Value" : Real AT %DB5070.DBD152, 500 ms
   "2925RS001A01T04.FP_PARAM.AuxLimit_L1_Value" : Real AT %DB5070.DBD156, 500 ms
   "2925RS001A01T04.Unit" : TextRef, internal   // Еденицы измерения При експорте из ECS через скрипт заполняется автоматически, если теги копируются в ручную то требуется задатать свойство Text
   "2925RS001A01T04.Decimals" : TextRef, internal   // Формат отображения При експорте из ECS через скрипт, заполняется автоматически. Если теги копируются в ручную то требуется задатать свойство Text s999999.9
   "2925RS001A01T04.FP_EN.Square" : Bool AT %DB5070.DBX46.0, 500 ms
   "2925RS001A01T04.FP_EN.SquareRoot" : Bool AT %DB5070.DBX46.1, 500 ms
   "2925RS001A01T04.FP_EN.ParentSupress" : Bool AT %DB5070.DBX46.2, 500 ms
   "2925RS001A01T04.FP_EN.ParentSupressUnit" : Bool AT %DB5070.DBX46.3, 500 ms
   "2925RS001A01T04.FP_EN.Force" : Bool AT %DB5070.DBX46.4, 500 ms
   "2925RS001A01T04.FP_EN.Damping" : Bool AT %DB5070.DBX46.5, 500 ms
   "2925RS001A01T04.FP_EN.Gradient_Pos" : Bool AT %DB5070.DBX46.6, 500 ms
   "2925RS001A01T04.FP_EN.Gradient_Neg" : Bool AT %DB5070.DBX46.7, 500 ms
   "2925RS001A01T04.FP_EN.Hysteresis" : Bool AT %DB5070.DBX47.0, 500 ms
   "2925RS001A01T04.FP_EN.Alarm_H3" : Bool AT %DB5070.DBX47.1, 500 ms
   "2925RS001A01T04.FP_EN.Alarm_H2" : Bool AT %DB5070.DBX47.2, 500 ms
   "2925RS001A01T04.FP_EN.Alarm_H1" : Bool AT %DB5070.DBX47.3, 500 ms
   "2925RS001A01T04.FP_EN.Alarm_L1" : Bool AT %DB5070.DBX47.4, 500 ms
   "2925RS001A01T04.FP_EN.Alarm_L2" : Bool AT %DB5070.DBX47.5, 500 ms
   "2925RS001A01T04.FP_EN.Alarm_L3" : Bool AT %DB5070.DBX47.6, 500 ms
   "2925RS001A01T04.FP_EN.AlarmDelay_H3" : Bool AT %DB5070.DBX47.7, 500 ms
   "2925RS001A01T04.FP_EN.AlarmDelay_H2" : Bool AT %DB5070.DBX48.0, 500 ms
   "2925RS001A01T04.FP_EN.AlarmDelay_H1" : Bool AT %DB5070.DBX48.1, 500 ms
   "2925RS001A01T04.FP_EN.AlarmDelay_L1" : Bool AT %DB5070.DBX48.2, 500 ms
   "2925RS001A01T04.FP_EN.AlarmDelay_L2" : Bool AT %DB5070.DBX48.3, 500 ms
   "2925RS001A01T04.FP_EN.AlarmDelay_L3" : Bool AT %DB5070.DBX48.4, 500 ms
   "2925RS001A01T04.FP_EN.ROC_Warn" : Bool AT %DB5070.DBX48.5, 500 ms
   "2925RS001A01T04.FP_EN.U_Range_Warn" : Bool AT %DB5070.DBX48.6, 500 ms
   "2925RS001A01T04.FP_EN.O_Range_Warn" : Bool AT %DB5070.DBX48.7, 500 ms
   "2925RS001A01T04.trend_tag_name" : TextRef, internal   // Еденицы измерения При експорте из ECS через скрипт - заполняется автоматически, если теги копируются в ручную то требуется задатать свойство Text - имя тега для тренда
   "2925RS001A01T04.DQ.AL_H3" : Bool AT %DB5070.DBX16.0, 500 ms
   "2925RS001A01T04.DQ.AL_H2" : Bool AT %DB5070.DBX16.1, 500 ms
   "2925RS001A01T04.DQ.AL_H1" : Bool AT %DB5070.DBX16.2, 500 ms
   "2925RS001A01T04.DQ.AL_L1" : Bool AT %DB5070.DBX16.3, 500 ms
   "2925RS001A01T04.DQ.AL_L2" : Bool AT %DB5070.DBX16.4, 500 ms
   "2925RS001A01T04.DQ.AL_L3" : Bool AT %DB5070.DBX16.5, 500 ms
   "2925RS001A01T04.DQ.SIG_OK" : Bool AT %DB5070.DBX16.6, 500 ms
   "2925RS001A01T04.DQ.LIM_H2" : Bool AT %DB5070.DBX16.7, 500 ms
   "2925RS001A01T04.DQ.LIM_H1" : Bool AT %DB5070.DBX17.0, 500 ms
   "2925RS001A01T04.DQ.LIM_L1" : Bool AT %DB5070.DBX17.1, 500 ms
   "2925RS001A01T04.DQ.LIM_L2" : Bool AT %DB5070.DBX17.2, 500 ms
   "2925RS001A01T04.DQ.GR_P" : Bool AT %DB5070.DBX17.3, 500 ms
   "2925RS001A01T04.DQ.GR_N" : Bool AT %DB5070.DBX17.4, 500 ms
   "2925RS001A01T04.I.IN" : Real AT %DB5070.DBD2, 500 ms
   "2925RS001A01T04.I.SIG_TYPE" : Int AT %DB5070.DBW0, 500 ms
   "2925RS001A01T04.I.FI_BUS" : Byte AT %DB5070.DBB6, 500 ms
   "2925RS001A01T04.DI.U_RANGE" : Bool AT %DB5070.DBX7.0, 500 ms
   "2925RS001A01T04.DI.O_RANGE" : Bool AT %DB5070.DBX7.1, 500 ms
   "2925RS001A01T04.DI.SIG_FAULT" : Bool AT %DB5070.DBX7.2, 500 ms
   "2925RS001A01T04.DI.EnConfig" : Bool AT %DB5070.DBX7.3, 500 ms
   "2925RS001A01T04.DI.AEN" : Bool AT %DB5070.DBX7.4, 500 ms
   "2925RS001A01T04.DI.AL_SUPR" : Bool AT %DB5070.DBX7.5, 500 ms
   "2925RS001A01T04.Q.PV_NORM" : Real AT %DB5070.DBD8, 500 ms
   "2925RS001A01T04.Q.PV_SCAL" : Real AT %DB5070.DBD12, 500 ms
   "2925RS001A01T04.ParentInfo" : TextRef, internal   // Имя родителя для попап окна, вкладка инфо. При експорте из ECS через скрипт заполняется автоматически, если теги копируются в ручную то требуется в ручную задатать свойство Start Value

HMI tags "2925RS001A01T05"
   "2925RS001A01T05.MSW" : 52809b66-421d-457f-8884-6f7a49d4e247 AT %DB5071.DBX18.0, 500 ms
   "2925RS001A01T05.DefaultText" : TextRef, internal   // Заголовок POPUP окна. При експорте из ECS через скрипт заполняется автоматически, если теги копируются в ручную то требуется в ручную задатать свойство Start Value
   "2925RS001A01T05.BlockInfo" : Array [0..2] of Int AT %DB5071.DBX38.0, 500 ms
   "2925RS001A01T05.StatusWork" : Int AT %DB5071.DBW242, 500 ms
   "2925RS001A01T05.FP_PARAM.DampingTime" : Int AT %DB5071.DBW50, 500 ms
   "2925RS001A01T05.FP_PARAM.Force_Value" : Real AT %DB5071.DBD52, 500 ms
   "2925RS001A01T05.FP_PARAM.Scale_Min" : Real AT %DB5071.DBD56, 500 ms
   "2925RS001A01T05.FP_PARAM.Scale_Max" : Real AT %DB5071.DBD60, 500 ms
   "2925RS001A01T05.FP_PARAM.Gradient" : Real AT %DB5071.DBD64, 500 ms
   "2925RS001A01T05.FP_PARAM.Grad_Pos" : Real AT %DB5071.DBD68, 500 ms
   "2925RS001A01T05.FP_PARAM.Grad_Neg" : Real AT %DB5071.DBD72, 500 ms
   "2925RS001A01T05.FP_PARAM.Grad_X" : Real AT %DB5071.DBD76, 500 ms
   "2925RS001A01T05.FP_PARAM.Gradient_Time_Pre" : Int AT %DB5071.DBW80, 500 ms
   "2925RS001A01T05.FP_PARAM.Gradient_Time_ACC" : Int AT %DB5071.DBW82, 500 ms
   "2925RS001A01T05.FP_PARAM.Alarm_Hyst" : Real AT %DB5071.DBD84, 500 ms
   "2925RS001A01T05.FP_PARAM.AlarmLimit_H3" : Real AT %DB5071.DBD88, 500 ms
   "2925RS001A01T05.FP_PARAM.AlarmLimit_H2" : Real AT %DB5071.DBD92, 500 ms
   "2925RS001A01T05.FP_PARAM.AlarmLimit_H1" : Real AT %DB5071.DBD96, 500 ms
   "2925RS001A01T05.FP_PARAM.AlarmLimit_L1" : Real AT %DB5071.DBD100, 500 ms
   "2925RS001A01T05.FP_PARAM.AlarmLimit_L2" : Real AT %DB5071.DBD104, 500 ms
   "2925RS001A01T05.FP_PARAM.AlarmLimit_L3" : Real AT %DB5071.DBD108, 500 ms
   "2925RS001A01T05.FP_PARAM.AlarmDelay_H3_Pre" : Int AT %DB5071.DBW112, 500 ms
   "2925RS001A01T05.FP_PARAM.AlarmDelay_H3_Acc" : Int AT %DB5071.DBW114, 500 ms
   "2925RS001A01T05.FP_PARAM.AlarmDelay_H2_Pre" : Int AT %DB5071.DBW116, 500 ms
   "2925RS001A01T05.FP_PARAM.AlarmDelay_H2_Acc" : Int AT %DB5071.DBW118, 500 ms
   "2925RS001A01T05.FP_PARAM.AlarmDelay_H1_Pre" : Int AT %DB5071.DBW120, 500 ms
   "2925RS001A01T05.FP_PARAM.AlarmDelay_H1_Acc" : Int AT %DB5071.DBW122, 500 ms
   "2925RS001A01T05.FP_PARAM.AlarmDelay_L1_Pre" : Int AT %DB5071.DBW124, 500 ms
   "2925RS001A01T05.FP_PARAM.AlarmDelay_L1_Acc" : Int AT %DB5071.DBW126, 500 ms
   "2925RS001A01T05.FP_PARAM.AlarmDelay_L2_Pre" : Int AT %DB5071.DBW128, 500 ms
   "2925RS001A01T05.FP_PARAM.AlarmDelay_L2_Acc" : Int AT %DB5071.DBW130, 500 ms
   "2925RS001A01T05.FP_PARAM.AlarmDelay_L3_Pre" : Int AT %DB5071.DBW132, 500 ms
   "2925RS001A01T05.FP_PARAM.AlarmDelay_L3_Acc" : Int AT %DB5071.DBW134, 500 ms
   "2925RS001A01T05.FP_PARAM.OpenLoopDelay_Pre" : Int AT %DB5071.DBW136, 500 ms
   "2925RS001A01T05.FP_PARAM.OpenLoopDelay_Acc" : Int AT %DB5071.DBW138, 500 ms
   "2925RS001A01T05.FP_PARAM.OverRangeDelay_Pre" : Int AT %DB5071.DBW140, 500 ms
   "2925RS001A01T05.FP_PARAM.OverRangeDelay_Acc" : Int AT %DB5071.DBW142, 500 ms
   "2925RS001A01T05.FP_PARAM.AuxLimit_H2_Value" : Real AT %DB5071.DBD144, 500 ms
   "2925RS001A01T05.FP_PARAM.AuxLimit_H1_Value" : Real AT %DB5071.DBD148, 500 ms
   "2925RS001A01T05.FP_PARAM.AuxLimit_L2_Value" : Real AT %DB5071.DBD152, 500 ms
   "2925RS001A01T05.FP_PARAM.AuxLimit_L1_Value" : Real AT %DB5071.DBD156, 500 ms
   "2925RS001A01T05.Unit" : TextRef, internal   // Еденицы измерения При експорте из ECS через скрипт заполняется автоматически, если теги копируются в ручную то требуется задатать свойство Text
   "2925RS001A01T05.Decimals" : TextRef, internal   // Формат отображения При експорте из ECS через скрипт, заполняется автоматически. Если теги копируются в ручную то требуется задатать свойство Text s999999.9
   "2925RS001A01T05.FP_EN.Square" : Bool AT %DB5071.DBX46.0, 500 ms
   "2925RS001A01T05.FP_EN.SquareRoot" : Bool AT %DB5071.DBX46.1, 500 ms
   "2925RS001A01T05.FP_EN.ParentSupress" : Bool AT %DB5071.DBX46.2, 500 ms
   "2925RS001A01T05.FP_EN.ParentSupressUnit" : Bool AT %DB5071.DBX46.3, 500 ms
   "2925RS001A01T05.FP_EN.Force" : Bool AT %DB5071.DBX46.4, 500 ms
   "2925RS001A01T05.FP_EN.Damping" : Bool AT %DB5071.DBX46.5, 500 ms
   "2925RS001A01T05.FP_EN.Gradient_Pos" : Bool AT %DB5071.DBX46.6, 500 ms
   "2925RS001A01T05.FP_EN.Gradient_Neg" : Bool AT %DB5071.DBX46.7, 500 ms
   "2925RS001A01T05.FP_EN.Hysteresis" : Bool AT %DB5071.DBX47.0, 500 ms
   "2925RS001A01T05.FP_EN.Alarm_H3" : Bool AT %DB5071.DBX47.1, 500 ms
   "2925RS001A01T05.FP_EN.Alarm_H2" : Bool AT %DB5071.DBX47.2, 500 ms
   "2925RS001A01T05.FP_EN.Alarm_H1" : Bool AT %DB5071.DBX47.3, 500 ms
   "2925RS001A01T05.FP_EN.Alarm_L1" : Bool AT %DB5071.DBX47.4, 500 ms
   "2925RS001A01T05.FP_EN.Alarm_L2" : Bool AT %DB5071.DBX47.5, 500 ms
   "2925RS001A01T05.FP_EN.Alarm_L3" : Bool AT %DB5071.DBX47.6, 500 ms
   "2925RS001A01T05.FP_EN.AlarmDelay_H3" : Bool AT %DB5071.DBX47.7, 500 ms
   "2925RS001A01T05.FP_EN.AlarmDelay_H2" : Bool AT %DB5071.DBX48.0, 500 ms
   "2925RS001A01T05.FP_EN.AlarmDelay_H1" : Bool AT %DB5071.DBX48.1, 500 ms
   "2925RS001A01T05.FP_EN.AlarmDelay_L1" : Bool AT %DB5071.DBX48.2, 500 ms
   "2925RS001A01T05.FP_EN.AlarmDelay_L2" : Bool AT %DB5071.DBX48.3, 500 ms
   "2925RS001A01T05.FP_EN.AlarmDelay_L3" : Bool AT %DB5071.DBX48.4, 500 ms
   "2925RS001A01T05.FP_EN.ROC_Warn" : Bool AT %DB5071.DBX48.5, 500 ms
   "2925RS001A01T05.FP_EN.U_Range_Warn" : Bool AT %DB5071.DBX48.6, 500 ms
   "2925RS001A01T05.FP_EN.O_Range_Warn" : Bool AT %DB5071.DBX48.7, 500 ms
   "2925RS001A01T05.trend_tag_name" : TextRef, internal   // Еденицы измерения При експорте из ECS через скрипт - заполняется автоматически, если теги копируются в ручную то требуется задатать свойство Text - имя тега для тренда
   "2925RS001A01T05.DQ.AL_H3" : Bool AT %DB5071.DBX16.0, 500 ms
   "2925RS001A01T05.DQ.AL_H2" : Bool AT %DB5071.DBX16.1, 500 ms
   "2925RS001A01T05.DQ.AL_H1" : Bool AT %DB5071.DBX16.2, 500 ms
   "2925RS001A01T05.DQ.AL_L1" : Bool AT %DB5071.DBX16.3, 500 ms
   "2925RS001A01T05.DQ.AL_L2" : Bool AT %DB5071.DBX16.4, 500 ms
   "2925RS001A01T05.DQ.AL_L3" : Bool AT %DB5071.DBX16.5, 500 ms
   "2925RS001A01T05.DQ.SIG_OK" : Bool AT %DB5071.DBX16.6, 500 ms
   "2925RS001A01T05.DQ.LIM_H2" : Bool AT %DB5071.DBX16.7, 500 ms
   "2925RS001A01T05.DQ.LIM_H1" : Bool AT %DB5071.DBX17.0, 500 ms
   "2925RS001A01T05.DQ.LIM_L1" : Bool AT %DB5071.DBX17.1, 500 ms
   "2925RS001A01T05.DQ.LIM_L2" : Bool AT %DB5071.DBX17.2, 500 ms
   "2925RS001A01T05.DQ.GR_P" : Bool AT %DB5071.DBX17.3, 500 ms
   "2925RS001A01T05.DQ.GR_N" : Bool AT %DB5071.DBX17.4, 500 ms
   "2925RS001A01T05.I.IN" : Real AT %DB5071.DBD2, 500 ms
   "2925RS001A01T05.I.SIG_TYPE" : Int AT %DB5071.DBW0, 500 ms
   "2925RS001A01T05.I.FI_BUS" : Byte AT %DB5071.DBB6, 500 ms
   "2925RS001A01T05.DI.U_RANGE" : Bool AT %DB5071.DBX7.0, 500 ms
   "2925RS001A01T05.DI.O_RANGE" : Bool AT %DB5071.DBX7.1, 500 ms
   "2925RS001A01T05.DI.SIG_FAULT" : Bool AT %DB5071.DBX7.2, 500 ms
   "2925RS001A01T05.DI.EnConfig" : Bool AT %DB5071.DBX7.3, 500 ms
   "2925RS001A01T05.DI.AEN" : Bool AT %DB5071.DBX7.4, 500 ms
   "2925RS001A01T05.DI.AL_SUPR" : Bool AT %DB5071.DBX7.5, 500 ms
   "2925RS001A01T05.Q.PV_NORM" : Real AT %DB5071.DBD8, 500 ms
   "2925RS001A01T05.Q.PV_SCAL" : Real AT %DB5071.DBD12, 500 ms
   "2925RS001A01T05.ParentInfo" : TextRef, internal   // Имя родителя для попап окна, вкладка инфо. При експорте из ECS через скрипт заполняется автоматически, если теги копируются в ручную то требуется в ручную задатать свойство Start Value

HMI tags "2930RS001A01F01"
   "2930RS001A01F01.MSW" : 52809b66-421d-457f-8884-6f7a49d4e247 AT %DB5086.DBX18.0, 500 ms
   "2930RS001A01F01.DefaultText" : TextRef, internal   // Заголовок POPUP окна. При експорте из ECS через скрипт заполняется автоматически, если теги копируются в ручную то требуется в ручную задатать свойство Start Value
   "2930RS001A01F01.BlockInfo" : Array [0..2] of Int AT %DB5086.DBX38.0, 500 ms
   "2930RS001A01F01.StatusWork" : Int AT %DB5086.DBW242, 500 ms
   "2930RS001A01F01.FP_PARAM.DampingTime" : Int AT %DB5086.DBW50, 500 ms
   "2930RS001A01F01.FP_PARAM.Force_Value" : Real AT %DB5086.DBD52, 500 ms
   "2930RS001A01F01.FP_PARAM.Scale_Min" : Real AT %DB5086.DBD56, 500 ms
   "2930RS001A01F01.FP_PARAM.Scale_Max" : Real AT %DB5086.DBD60, 500 ms
   "2930RS001A01F01.FP_PARAM.Gradient" : Real AT %DB5086.DBD64, 500 ms
   "2930RS001A01F01.FP_PARAM.Grad_Pos" : Real AT %DB5086.DBD68, 500 ms
   "2930RS001A01F01.FP_PARAM.Grad_Neg" : Real AT %DB5086.DBD72, 500 ms
   "2930RS001A01F01.FP_PARAM.Grad_X" : Real AT %DB5086.DBD76, 500 ms
   "2930RS001A01F01.FP_PARAM.Gradient_Time_Pre" : Int AT %DB5086.DBW80, 500 ms
   "2930RS001A01F01.FP_PARAM.Gradient_Time_ACC" : Int AT %DB5086.DBW82, 500 ms
   "2930RS001A01F01.FP_PARAM.Alarm_Hyst" : Real AT %DB5086.DBD84, 500 ms
   "2930RS001A01F01.FP_PARAM.AlarmLimit_H3" : Real AT %DB5086.DBD88, 500 ms
   "2930RS001A01F01.FP_PARAM.AlarmLimit_H2" : Real AT %DB5086.DBD92, 500 ms
   "2930RS001A01F01.FP_PARAM.AlarmLimit_H1" : Real AT %DB5086.DBD96, 500 ms
   "2930RS001A01F01.FP_PARAM.AlarmLimit_L1" : Real AT %DB5086.DBD100, 500 ms
   "2930RS001A01F01.FP_PARAM.AlarmLimit_L2" : Real AT %DB5086.DBD104, 500 ms
   "2930RS001A01F01.FP_PARAM.AlarmLimit_L3" : Real AT %DB5086.DBD108, 500 ms
   "2930RS001A01F01.FP_PARAM.AlarmDelay_H3_Pre" : Int AT %DB5086.DBW112, 500 ms
   "2930RS001A01F01.FP_PARAM.AlarmDelay_H3_Acc" : Int AT %DB5086.DBW114, 500 ms
   "2930RS001A01F01.FP_PARAM.AlarmDelay_H2_Pre" : Int AT %DB5086.DBW116, 500 ms
   "2930RS001A01F01.FP_PARAM.AlarmDelay_H2_Acc" : Int AT %DB5086.DBW118, 500 ms
   "2930RS001A01F01.FP_PARAM.AlarmDelay_H1_Pre" : Int AT %DB5086.DBW120, 500 ms
   "2930RS001A01F01.FP_PARAM.AlarmDelay_H1_Acc" : Int AT %DB5086.DBW122, 500 ms
   "2930RS001A01F01.FP_PARAM.AlarmDelay_L1_Pre" : Int AT %DB5086.DBW124, 500 ms
   "2930RS001A01F01.FP_PARAM.AlarmDelay_L1_Acc" : Int AT %DB5086.DBW126, 500 ms
   "2930RS001A01F01.FP_PARAM.AlarmDelay_L2_Pre" : Int AT %DB5086.DBW128, 500 ms
   "2930RS001A01F01.FP_PARAM.AlarmDelay_L2_Acc" : Int AT %DB5086.DBW130, 500 ms
   "2930RS001A01F01.FP_PARAM.AlarmDelay_L3_Pre" : Int AT %DB5086.DBW132, 500 ms
   "2930RS001A01F01.FP_PARAM.AlarmDelay_L3_Acc" : Int AT %DB5086.DBW134, 500 ms
   "2930RS001A01F01.FP_PARAM.OpenLoopDelay_Pre" : Int AT %DB5086.DBW136, 500 ms
   "2930RS001A01F01.FP_PARAM.OpenLoopDelay_Acc" : Int AT %DB5086.DBW138, 500 ms
   "2930RS001A01F01.FP_PARAM.OverRangeDelay_Pre" : Int AT %DB5086.DBW140, 500 ms
   "2930RS001A01F01.FP_PARAM.OverRangeDelay_Acc" : Int AT %DB5086.DBW142, 500 ms
   "2930RS001A01F01.FP_PARAM.AuxLimit_H2_Value" : Real AT %DB5086.DBD144, 500 ms
   "2930RS001A01F01.FP_PARAM.AuxLimit_H1_Value" : Real AT %DB5086.DBD148, 500 ms
   "2930RS001A01F01.FP_PARAM.AuxLimit_L2_Value" : Real AT %DB5086.DBD152, 500 ms
   "2930RS001A01F01.FP_PARAM.AuxLimit_L1_Value" : Real AT %DB5086.DBD156, 500 ms
   "2930RS001A01F01.Unit" : TextRef, internal   // Еденицы измерения При експорте из ECS через скрипт заполняется автоматически, если теги копируются в ручную то требуется задатать свойство Text
   "2930RS001A01F01.Decimals" : TextRef, internal   // Формат отображения При експорте из ECS через скрипт, заполняется автоматически. Если теги копируются в ручную то требуется задатать свойство Text s999999.9
   "2930RS001A01F01.FP_EN.Square" : Bool AT %DB5086.DBX46.0, 500 ms
   "2930RS001A01F01.FP_EN.SquareRoot" : Bool AT %DB5086.DBX46.1, 500 ms
   "2930RS001A01F01.FP_EN.ParentSupress" : Bool AT %DB5086.DBX46.2, 500 ms
   "2930RS001A01F01.FP_EN.ParentSupressUnit" : Bool AT %DB5086.DBX46.3, 500 ms
   "2930RS001A01F01.FP_EN.Force" : Bool AT %DB5086.DBX46.4, 500 ms
   "2930RS001A01F01.FP_EN.Damping" : Bool AT %DB5086.DBX46.5, 500 ms
   "2930RS001A01F01.FP_EN.Gradient_Pos" : Bool AT %DB5086.DBX46.6, 500 ms
   "2930RS001A01F01.FP_EN.Gradient_Neg" : Bool AT %DB5086.DBX46.7, 500 ms
   "2930RS001A01F01.FP_EN.Hysteresis" : Bool AT %DB5086.DBX47.0, 500 ms
   "2930RS001A01F01.FP_EN.Alarm_H3" : Bool AT %DB5086.DBX47.1, 500 ms
   "2930RS001A01F01.FP_EN.Alarm_H2" : Bool AT %DB5086.DBX47.2, 500 ms
   "2930RS001A01F01.FP_EN.Alarm_H1" : Bool AT %DB5086.DBX47.3, 500 ms
   "2930RS001A01F01.FP_EN.Alarm_L1" : Bool AT %DB5086.DBX47.4, 500 ms
   "2930RS001A01F01.FP_EN.Alarm_L2" : Bool AT %DB5086.DBX47.5, 500 ms
   "2930RS001A01F01.FP_EN.Alarm_L3" : Bool AT %DB5086.DBX47.6, 500 ms
   "2930RS001A01F01.FP_EN.AlarmDelay_H3" : Bool AT %DB5086.DBX47.7, 500 ms
   "2930RS001A01F01.FP_EN.AlarmDelay_H2" : Bool AT %DB5086.DBX48.0, 500 ms
   "2930RS001A01F01.FP_EN.AlarmDelay_H1" : Bool AT %DB5086.DBX48.1, 500 ms
   "2930RS001A01F01.FP_EN.AlarmDelay_L1" : Bool AT %DB5086.DBX48.2, 500 ms
   "2930RS001A01F01.FP_EN.AlarmDelay_L2" : Bool AT %DB5086.DBX48.3, 500 ms
   "2930RS001A01F01.FP_EN.AlarmDelay_L3" : Bool AT %DB5086.DBX48.4, 500 ms
   "2930RS001A01F01.FP_EN.ROC_Warn" : Bool AT %DB5086.DBX48.5, 500 ms
   "2930RS001A01F01.FP_EN.U_Range_Warn" : Bool AT %DB5086.DBX48.6, 500 ms
   "2930RS001A01F01.FP_EN.O_Range_Warn" : Bool AT %DB5086.DBX48.7, 500 ms
   "2930RS001A01F01.trend_tag_name" : TextRef, internal   // Еденицы измерения При експорте из ECS через скрипт - заполняется автоматически, если теги копируются в ручную то требуется задатать свойство Text - имя тега для тренда
   "2930RS001A01F01.DQ.AL_H3" : Bool AT %DB5086.DBX16.0, 500 ms
   "2930RS001A01F01.DQ.AL_H2" : Bool AT %DB5086.DBX16.1, 500 ms
   "2930RS001A01F01.DQ.AL_H1" : Bool AT %DB5086.DBX16.2, 500 ms
   "2930RS001A01F01.DQ.AL_L1" : Bool AT %DB5086.DBX16.3, 500 ms
   "2930RS001A01F01.DQ.AL_L2" : Bool AT %DB5086.DBX16.4, 500 ms
   "2930RS001A01F01.DQ.AL_L3" : Bool AT %DB5086.DBX16.5, 500 ms
   "2930RS001A01F01.DQ.SIG_OK" : Bool AT %DB5086.DBX16.6, 500 ms
   "2930RS001A01F01.DQ.LIM_H2" : Bool AT %DB5086.DBX16.7, 500 ms
   "2930RS001A01F01.DQ.LIM_H1" : Bool AT %DB5086.DBX17.0, 500 ms
   "2930RS001A01F01.DQ.LIM_L1" : Bool AT %DB5086.DBX17.1, 500 ms
   "2930RS001A01F01.DQ.LIM_L2" : Bool AT %DB5086.DBX17.2, 500 ms
   "2930RS001A01F01.DQ.GR_P" : Bool AT %DB5086.DBX17.3, 500 ms
   "2930RS001A01F01.DQ.GR_N" : Bool AT %DB5086.DBX17.4, 500 ms
   "2930RS001A01F01.I.IN" : Real AT %DB5086.DBD2, 500 ms
   "2930RS001A01F01.I.SIG_TYPE" : Int AT %DB5086.DBW0, 500 ms
   "2930RS001A01F01.I.FI_BUS" : Byte AT %DB5086.DBB6, 500 ms
   "2930RS001A01F01.DI.U_RANGE" : Bool AT %DB5086.DBX7.0, 500 ms
   "2930RS001A01F01.DI.O_RANGE" : Bool AT %DB5086.DBX7.1, 500 ms
   "2930RS001A01F01.DI.SIG_FAULT" : Bool AT %DB5086.DBX7.2, 500 ms
   "2930RS001A01F01.DI.EnConfig" : Bool AT %DB5086.DBX7.3, 500 ms
   "2930RS001A01F01.DI.AEN" : Bool AT %DB5086.DBX7.4, 500 ms
   "2930RS001A01F01.DI.AL_SUPR" : Bool AT %DB5086.DBX7.5, 500 ms
   "2930RS001A01F01.Q.PV_NORM" : Real AT %DB5086.DBD8, 500 ms
   "2930RS001A01F01.Q.PV_SCAL" : Real AT %DB5086.DBD12, 500 ms
   "2930RS001A01F01.ParentInfo" : TextRef, internal   // Имя родителя для попап окна, вкладка инфо. При експорте из ECS через скрипт заполняется автоматически, если теги копируются в ручную то требуется в ручную задатать свойство Start Value

HMI tags "2930RS001A01F02"
   "2930RS001A01F02.MSW" : 52809b66-421d-457f-8884-6f7a49d4e247 AT %DB5087.DBX18.0, 500 ms
   "2930RS001A01F02.DefaultText" : TextRef, internal   // Заголовок POPUP окна. При експорте из ECS через скрипт заполняется автоматически, если теги копируются в ручную то требуется в ручную задатать свойство Start Value
   "2930RS001A01F02.BlockInfo" : Array [0..2] of Int AT %DB5087.DBX38.0, 500 ms
   "2930RS001A01F02.StatusWork" : Int AT %DB5087.DBW242, 500 ms
   "2930RS001A01F02.FP_PARAM.DampingTime" : Int AT %DB5087.DBW50, 500 ms
   "2930RS001A01F02.FP_PARAM.Force_Value" : Real AT %DB5087.DBD52, 500 ms
   "2930RS001A01F02.FP_PARAM.Scale_Min" : Real AT %DB5087.DBD56, 500 ms
   "2930RS001A01F02.FP_PARAM.Scale_Max" : Real AT %DB5087.DBD60, 500 ms
   "2930RS001A01F02.FP_PARAM.Gradient" : Real AT %DB5087.DBD64, 500 ms
   "2930RS001A01F02.FP_PARAM.Grad_Pos" : Real AT %DB5087.DBD68, 500 ms
   "2930RS001A01F02.FP_PARAM.Grad_Neg" : Real AT %DB5087.DBD72, 500 ms
   "2930RS001A01F02.FP_PARAM.Grad_X" : Real AT %DB5087.DBD76, 500 ms
   "2930RS001A01F02.FP_PARAM.Gradient_Time_Pre" : Int AT %DB5087.DBW80, 500 ms
   "2930RS001A01F02.FP_PARAM.Gradient_Time_ACC" : Int AT %DB5087.DBW82, 500 ms
   "2930RS001A01F02.FP_PARAM.Alarm_Hyst" : Real AT %DB5087.DBD84, 500 ms
   "2930RS001A01F02.FP_PARAM.AlarmLimit_H3" : Real AT %DB5087.DBD88, 500 ms
   "2930RS001A01F02.FP_PARAM.AlarmLimit_H2" : Real AT %DB5087.DBD92, 500 ms
   "2930RS001A01F02.FP_PARAM.AlarmLimit_H1" : Real AT %DB5087.DBD96, 500 ms
   "2930RS001A01F02.FP_PARAM.AlarmLimit_L1" : Real AT %DB5087.DBD100, 500 ms
   "2930RS001A01F02.FP_PARAM.AlarmLimit_L2" : Real AT %DB5087.DBD104, 500 ms
   "2930RS001A01F02.FP_PARAM.AlarmLimit_L3" : Real AT %DB5087.DBD108, 500 ms
   "2930RS001A01F02.FP_PARAM.AlarmDelay_H3_Pre" : Int AT %DB5087.DBW112, 500 ms
   "2930RS001A01F02.FP_PARAM.AlarmDelay_H3_Acc" : Int AT %DB5087.DBW114, 500 ms
   "2930RS001A01F02.FP_PARAM.AlarmDelay_H2_Pre" : Int AT %DB5087.DBW116, 500 ms
   "2930RS001A01F02.FP_PARAM.AlarmDelay_H2_Acc" : Int AT %DB5087.DBW118, 500 ms
   "2930RS001A01F02.FP_PARAM.AlarmDelay_H1_Pre" : Int AT %DB5087.DBW120, 500 ms
   "2930RS001A01F02.FP_PARAM.AlarmDelay_H1_Acc" : Int AT %DB5087.DBW122, 500 ms
   "2930RS001A01F02.FP_PARAM.AlarmDelay_L1_Pre" : Int AT %DB5087.DBW124, 500 ms
   "2930RS001A01F02.FP_PARAM.AlarmDelay_L1_Acc" : Int AT %DB5087.DBW126, 500 ms
   "2930RS001A01F02.FP_PARAM.AlarmDelay_L2_Pre" : Int AT %DB5087.DBW128, 500 ms
   "2930RS001A01F02.FP_PARAM.AlarmDelay_L2_Acc" : Int AT %DB5087.DBW130, 500 ms
   "2930RS001A01F02.FP_PARAM.AlarmDelay_L3_Pre" : Int AT %DB5087.DBW132, 500 ms
   "2930RS001A01F02.FP_PARAM.AlarmDelay_L3_Acc" : Int AT %DB5087.DBW134, 500 ms
   "2930RS001A01F02.FP_PARAM.OpenLoopDelay_Pre" : Int AT %DB5087.DBW136, 500 ms
   "2930RS001A01F02.FP_PARAM.OpenLoopDelay_Acc" : Int AT %DB5087.DBW138, 500 ms
   "2930RS001A01F02.FP_PARAM.OverRangeDelay_Pre" : Int AT %DB5087.DBW140, 500 ms
   "2930RS001A01F02.FP_PARAM.OverRangeDelay_Acc" : Int AT %DB5087.DBW142, 500 ms
   "2930RS001A01F02.FP_PARAM.AuxLimit_H2_Value" : Real AT %DB5087.DBD144, 500 ms
   "2930RS001A01F02.FP_PARAM.AuxLimit_H1_Value" : Real AT %DB5087.DBD148, 500 ms
   "2930RS001A01F02.FP_PARAM.AuxLimit_L2_Value" : Real AT %DB5087.DBD152, 500 ms
   "2930RS001A01F02.FP_PARAM.AuxLimit_L1_Value" : Real AT %DB5087.DBD156, 500 ms
   "2930RS001A01F02.Unit" : TextRef, internal   // Еденицы измерения При експорте из ECS через скрипт заполняется автоматически, если теги копируются в ручную то требуется задатать свойство Text
   "2930RS001A01F02.Decimals" : TextRef, internal   // Формат отображения При експорте из ECS через скрипт, заполняется автоматически. Если теги копируются в ручную то требуется задатать свойство Text s999999.9
   "2930RS001A01F02.FP_EN.Square" : Bool AT %DB5087.DBX46.0, 500 ms
   "2930RS001A01F02.FP_EN.SquareRoot" : Bool AT %DB5087.DBX46.1, 500 ms
   "2930RS001A01F02.FP_EN.ParentSupress" : Bool AT %DB5087.DBX46.2, 500 ms
   "2930RS001A01F02.FP_EN.ParentSupressUnit" : Bool AT %DB5087.DBX46.3, 500 ms
   "2930RS001A01F02.FP_EN.Force" : Bool AT %DB5087.DBX46.4, 500 ms
   "2930RS001A01F02.FP_EN.Damping" : Bool AT %DB5087.DBX46.5, 500 ms
   "2930RS001A01F02.FP_EN.Gradient_Pos" : Bool AT %DB5087.DBX46.6, 500 ms
   "2930RS001A01F02.FP_EN.Gradient_Neg" : Bool AT %DB5087.DBX46.7, 500 ms
   "2930RS001A01F02.FP_EN.Hysteresis" : Bool AT %DB5087.DBX47.0, 500 ms
   "2930RS001A01F02.FP_EN.Alarm_H3" : Bool AT %DB5087.DBX47.1, 500 ms
   "2930RS001A01F02.FP_EN.Alarm_H2" : Bool AT %DB5087.DBX47.2, 500 ms
   "2930RS001A01F02.FP_EN.Alarm_H1" : Bool AT %DB5087.DBX47.3, 500 ms
   "2930RS001A01F02.FP_EN.Alarm_L1" : Bool AT %DB5087.DBX47.4, 500 ms
   "2930RS001A01F02.FP_EN.Alarm_L2" : Bool AT %DB5087.DBX47.5, 500 ms
   "2930RS001A01F02.FP_EN.Alarm_L3" : Bool AT %DB5087.DBX47.6, 500 ms
   "2930RS001A01F02.FP_EN.AlarmDelay_H3" : Bool AT %DB5087.DBX47.7, 500 ms
   "2930RS001A01F02.FP_EN.AlarmDelay_H2" : Bool AT %DB5087.DBX48.0, 500 ms
   "2930RS001A01F02.FP_EN.AlarmDelay_H1" : Bool AT %DB5087.DBX48.1, 500 ms
   "2930RS001A01F02.FP_EN.AlarmDelay_L1" : Bool AT %DB5087.DBX48.2, 500 ms
   "2930RS001A01F02.FP_EN.AlarmDelay_L2" : Bool AT %DB5087.DBX48.3, 500 ms
   "2930RS001A01F02.FP_EN.AlarmDelay_L3" : Bool AT %DB5087.DBX48.4, 500 ms
   "2930RS001A01F02.FP_EN.ROC_Warn" : Bool AT %DB5087.DBX48.5, 500 ms
   "2930RS001A01F02.FP_EN.U_Range_Warn" : Bool AT %DB5087.DBX48.6, 500 ms
   "2930RS001A01F02.FP_EN.O_Range_Warn" : Bool AT %DB5087.DBX48.7, 500 ms
   "2930RS001A01F02.trend_tag_name" : TextRef, internal   // Еденицы измерения При експорте из ECS через скрипт - заполняется автоматически, если теги копируются в ручную то требуется задатать свойство Text - имя тега для тренда
   "2930RS001A01F02.DQ.AL_H3" : Bool AT %DB5087.DBX16.0, 500 ms
   "2930RS001A01F02.DQ.AL_H2" : Bool AT %DB5087.DBX16.1, 500 ms
   "2930RS001A01F02.DQ.AL_H1" : Bool AT %DB5087.DBX16.2, 500 ms
   "2930RS001A01F02.DQ.AL_L1" : Bool AT %DB5087.DBX16.3, 500 ms
   "2930RS001A01F02.DQ.AL_L2" : Bool AT %DB5087.DBX16.4, 500 ms
   "2930RS001A01F02.DQ.AL_L3" : Bool AT %DB5087.DBX16.5, 500 ms
   "2930RS001A01F02.DQ.SIG_OK" : Bool AT %DB5087.DBX16.6, 500 ms
   "2930RS001A01F02.DQ.LIM_H2" : Bool AT %DB5087.DBX16.7, 500 ms
   "2930RS001A01F02.DQ.LIM_H1" : Bool AT %DB5087.DBX17.0, 500 ms
   "2930RS001A01F02.DQ.LIM_L1" : Bool AT %DB5087.DBX17.1, 500 ms
   "2930RS001A01F02.DQ.LIM_L2" : Bool AT %DB5087.DBX17.2, 500 ms
   "2930RS001A01F02.DQ.GR_P" : Bool AT %DB5087.DBX17.3, 500 ms
   "2930RS001A01F02.DQ.GR_N" : Bool AT %DB5087.DBX17.4, 500 ms
   "2930RS001A01F02.I.IN" : Real AT %DB5087.DBD2, 500 ms
   "2930RS001A01F02.I.SIG_TYPE" : Int AT %DB5087.DBW0, 500 ms
   "2930RS001A01F02.I.FI_BUS" : Byte AT %DB5087.DBB6, 500 ms
   "2930RS001A01F02.DI.U_RANGE" : Bool AT %DB5087.DBX7.0, 500 ms
   "2930RS001A01F02.DI.O_RANGE" : Bool AT %DB5087.DBX7.1, 500 ms
   "2930RS001A01F02.DI.SIG_FAULT" : Bool AT %DB5087.DBX7.2, 500 ms
   "2930RS001A01F02.DI.EnConfig" : Bool AT %DB5087.DBX7.3, 500 ms
   "2930RS001A01F02.DI.AEN" : Bool AT %DB5087.DBX7.4, 500 ms
   "2930RS001A01F02.DI.AL_SUPR" : Bool AT %DB5087.DBX7.5, 500 ms
   "2930RS001A01F02.Q.PV_NORM" : Real AT %DB5087.DBD8, 500 ms
   "2930RS001A01F02.Q.PV_SCAL" : Real AT %DB5087.DBD12, 500 ms
   "2930RS001A01F02.ParentInfo" : TextRef, internal   // Имя родителя для попап окна, вкладка инфо. При експорте из ECS через скрипт заполняется автоматически, если теги копируются в ручную то требуется в ручную задатать свойство Start Value

HMI tags "2930RS001A01F03"
   "2930RS001A01F03.MSW" : 52809b66-421d-457f-8884-6f7a49d4e247 AT %DB5088.DBX18.0, 500 ms
   "2930RS001A01F03.DefaultText" : TextRef, internal   // Заголовок POPUP окна. При експорте из ECS через скрипт заполняется автоматически, если теги копируются в ручную то требуется в ручную задатать свойство Start Value
   "2930RS001A01F03.BlockInfo" : Array [0..2] of Int AT %DB5088.DBX38.0, 500 ms
   "2930RS001A01F03.StatusWork" : Int AT %DB5088.DBW242, 500 ms
   "2930RS001A01F03.FP_PARAM.DampingTime" : Int AT %DB5088.DBW50, 500 ms
   "2930RS001A01F03.FP_PARAM.Force_Value" : Real AT %DB5088.DBD52, 500 ms
   "2930RS001A01F03.FP_PARAM.Scale_Min" : Real AT %DB5088.DBD56, 500 ms
   "2930RS001A01F03.FP_PARAM.Scale_Max" : Real AT %DB5088.DBD60, 500 ms
   "2930RS001A01F03.FP_PARAM.Gradient" : Real AT %DB5088.DBD64, 500 ms
   "2930RS001A01F03.FP_PARAM.Grad_Pos" : Real AT %DB5088.DBD68, 500 ms
   "2930RS001A01F03.FP_PARAM.Grad_Neg" : Real AT %DB5088.DBD72, 500 ms
   "2930RS001A01F03.FP_PARAM.Grad_X" : Real AT %DB5088.DBD76, 500 ms
   "2930RS001A01F03.FP_PARAM.Gradient_Time_Pre" : Int AT %DB5088.DBW80, 500 ms
   "2930RS001A01F03.FP_PARAM.Gradient_Time_ACC" : Int AT %DB5088.DBW82, 500 ms
   "2930RS001A01F03.FP_PARAM.Alarm_Hyst" : Real AT %DB5088.DBD84, 500 ms
   "2930RS001A01F03.FP_PARAM.AlarmLimit_H3" : Real AT %DB5088.DBD88, 500 ms
   "2930RS001A01F03.FP_PARAM.AlarmLimit_H2" : Real AT %DB5088.DBD92, 500 ms
   "2930RS001A01F03.FP_PARAM.AlarmLimit_H1" : Real AT %DB5088.DBD96, 500 ms
   "2930RS001A01F03.FP_PARAM.AlarmLimit_L1" : Real AT %DB5088.DBD100, 500 ms
   "2930RS001A01F03.FP_PARAM.AlarmLimit_L2" : Real AT %DB5088.DBD104, 500 ms
   "2930RS001A01F03.FP_PARAM.AlarmLimit_L3" : Real AT %DB5088.DBD108, 500 ms
   "2930RS001A01F03.FP_PARAM.AlarmDelay_H3_Pre" : Int AT %DB5088.DBW112, 500 ms
   "2930RS001A01F03.FP_PARAM.AlarmDelay_H3_Acc" : Int AT %DB5088.DBW114, 500 ms
   "2930RS001A01F03.FP_PARAM.AlarmDelay_H2_Pre" : Int AT %DB5088.DBW116, 500 ms
   "2930RS001A01F03.FP_PARAM.AlarmDelay_H2_Acc" : Int AT %DB5088.DBW118, 500 ms
   "2930RS001A01F03.FP_PARAM.AlarmDelay_H1_Pre" : Int AT %DB5088.DBW120, 500 ms
   "2930RS001A01F03.FP_PARAM.AlarmDelay_H1_Acc" : Int AT %DB5088.DBW122, 500 ms
   "2930RS001A01F03.FP_PARAM.AlarmDelay_L1_Pre" : Int AT %DB5088.DBW124, 500 ms
   "2930RS001A01F03.FP_PARAM.AlarmDelay_L1_Acc" : Int AT %DB5088.DBW126, 500 ms
   "2930RS001A01F03.FP_PARAM.AlarmDelay_L2_Pre" : Int AT %DB5088.DBW128, 500 ms
   "2930RS001A01F03.FP_PARAM.AlarmDelay_L2_Acc" : Int AT %DB5088.DBW130, 500 ms
   "2930RS001A01F03.FP_PARAM.AlarmDelay_L3_Pre" : Int AT %DB5088.DBW132, 500 ms
   "2930RS001A01F03.FP_PARAM.AlarmDelay_L3_Acc" : Int AT %DB5088.DBW134, 500 ms
   "2930RS001A01F03.FP_PARAM.OpenLoopDelay_Pre" : Int AT %DB5088.DBW136, 500 ms
   "2930RS001A01F03.FP_PARAM.OpenLoopDelay_Acc" : Int AT %DB5088.DBW138, 500 ms
   "2930RS001A01F03.FP_PARAM.OverRangeDelay_Pre" : Int AT %DB5088.DBW140, 500 ms
   "2930RS001A01F03.FP_PARAM.OverRangeDelay_Acc" : Int AT %DB5088.DBW142, 500 ms
   "2930RS001A01F03.FP_PARAM.AuxLimit_H2_Value" : Real AT %DB5088.DBD144, 500 ms
   "2930RS001A01F03.FP_PARAM.AuxLimit_H1_Value" : Real AT %DB5088.DBD148, 500 ms
   "2930RS001A01F03.FP_PARAM.AuxLimit_L2_Value" : Real AT %DB5088.DBD152, 500 ms
   "2930RS001A01F03.FP_PARAM.AuxLimit_L1_Value" : Real AT %DB5088.DBD156, 500 ms
   "2930RS001A01F03.Unit" : TextRef, internal   // Еденицы измерения При експорте из ECS через скрипт заполняется автоматически, если теги копируются в ручную то требуется задатать свойство Text
   "2930RS001A01F03.Decimals" : TextRef, internal   // Формат отображения При експорте из ECS через скрипт, заполняется автоматически. Если теги копируются в ручную то требуется задатать свойство Text s999999.9
   "2930RS001A01F03.FP_EN.Square" : Bool AT %DB5088.DBX46.0, 500 ms
   "2930RS001A01F03.FP_EN.SquareRoot" : Bool AT %DB5088.DBX46.1, 500 ms
   "2930RS001A01F03.FP_EN.ParentSupress" : Bool AT %DB5088.DBX46.2, 500 ms
   "2930RS001A01F03.FP_EN.ParentSupressUnit" : Bool AT %DB5088.DBX46.3, 500 ms
   "2930RS001A01F03.FP_EN.Force" : Bool AT %DB5088.DBX46.4, 500 ms
   "2930RS001A01F03.FP_EN.Damping" : Bool AT %DB5088.DBX46.5, 500 ms
   "2930RS001A01F03.FP_EN.Gradient_Pos" : Bool AT %DB5088.DBX46.6, 500 ms
   "2930RS001A01F03.FP_EN.Gradient_Neg" : Bool AT %DB5088.DBX46.7, 500 ms
   "2930RS001A01F03.FP_EN.Hysteresis" : Bool AT %DB5088.DBX47.0, 500 ms
   "2930RS001A01F03.FP_EN.Alarm_H3" : Bool AT %DB5088.DBX47.1, 500 ms
   "2930RS001A01F03.FP_EN.Alarm_H2" : Bool AT %DB5088.DBX47.2, 500 ms
   "2930RS001A01F03.FP_EN.Alarm_H1" : Bool AT %DB5088.DBX47.3, 500 ms
   "2930RS001A01F03.FP_EN.Alarm_L1" : Bool AT %DB5088.DBX47.4, 500 ms
   "2930RS001A01F03.FP_EN.Alarm_L2" : Bool AT %DB5088.DBX47.5, 500 ms
   "2930RS001A01F03.FP_EN.Alarm_L3" : Bool AT %DB5088.DBX47.6, 500 ms
   "2930RS001A01F03.FP_EN.AlarmDelay_H3" : Bool AT %DB5088.DBX47.7, 500 ms
   "2930RS001A01F03.FP_EN.AlarmDelay_H2" : Bool AT %DB5088.DBX48.0, 500 ms
   "2930RS001A01F03.FP_EN.AlarmDelay_H1" : Bool AT %DB5088.DBX48.1, 500 ms
   "2930RS001A01F03.FP_EN.AlarmDelay_L1" : Bool AT %DB5088.DBX48.2, 500 ms
   "2930RS001A01F03.FP_EN.AlarmDelay_L2" : Bool AT %DB5088.DBX48.3, 500 ms
   "2930RS001A01F03.FP_EN.AlarmDelay_L3" : Bool AT %DB5088.DBX48.4, 500 ms
   "2930RS001A01F03.FP_EN.ROC_Warn" : Bool AT %DB5088.DBX48.5, 500 ms
   "2930RS001A01F03.FP_EN.U_Range_Warn" : Bool AT %DB5088.DBX48.6, 500 ms
   "2930RS001A01F03.FP_EN.O_Range_Warn" : Bool AT %DB5088.DBX48.7, 500 ms
   "2930RS001A01F03.trend_tag_name" : TextRef, internal   // Еденицы измерения При експорте из ECS через скрипт - заполняется автоматически, если теги копируются в ручную то требуется задатать свойство Text - имя тега для тренда
   "2930RS001A01F03.DQ.AL_H3" : Bool AT %DB5088.DBX16.0, 500 ms
   "2930RS001A01F03.DQ.AL_H2" : Bool AT %DB5088.DBX16.1, 500 ms
   "2930RS001A01F03.DQ.AL_H1" : Bool AT %DB5088.DBX16.2, 500 ms
   "2930RS001A01F03.DQ.AL_L1" : Bool AT %DB5088.DBX16.3, 500 ms
   "2930RS001A01F03.DQ.AL_L2" : Bool AT %DB5088.DBX16.4, 500 ms
   "2930RS001A01F03.DQ.AL_L3" : Bool AT %DB5088.DBX16.5, 500 ms
   "2930RS001A01F03.DQ.SIG_OK" : Bool AT %DB5088.DBX16.6, 500 ms
   "2930RS001A01F03.DQ.LIM_H2" : Bool AT %DB5088.DBX16.7, 500 ms
   "2930RS001A01F03.DQ.LIM_H1" : Bool AT %DB5088.DBX17.0, 500 ms
   "2930RS001A01F03.DQ.LIM_L1" : Bool AT %DB5088.DBX17.1, 500 ms
   "2930RS001A01F03.DQ.LIM_L2" : Bool AT %DB5088.DBX17.2, 500 ms
   "2930RS001A01F03.DQ.GR_P" : Bool AT %DB5088.DBX17.3, 500 ms
   "2930RS001A01F03.DQ.GR_N" : Bool AT %DB5088.DBX17.4, 500 ms
   "2930RS001A01F03.I.IN" : Real AT %DB5088.DBD2, 500 ms
   "2930RS001A01F03.I.SIG_TYPE" : Int AT %DB5088.DBW0, 500 ms
   "2930RS001A01F03.I.FI_BUS" : Byte AT %DB5088.DBB6, 500 ms
   "2930RS001A01F03.DI.U_RANGE" : Bool AT %DB5088.DBX7.0, 500 ms
   "2930RS001A01F03.DI.O_RANGE" : Bool AT %DB5088.DBX7.1, 500 ms
   "2930RS001A01F03.DI.SIG_FAULT" : Bool AT %DB5088.DBX7.2, 500 ms
   "2930RS001A01F03.DI.EnConfig" : Bool AT %DB5088.DBX7.3, 500 ms
   "2930RS001A01F03.DI.AEN" : Bool AT %DB5088.DBX7.4, 500 ms
   "2930RS001A01F03.DI.AL_SUPR" : Bool AT %DB5088.DBX7.5, 500 ms
   "2930RS001A01F03.Q.PV_NORM" : Real AT %DB5088.DBD8, 500 ms
   "2930RS001A01F03.Q.PV_SCAL" : Real AT %DB5088.DBD12, 500 ms
   "2930RS001A01F03.ParentInfo" : TextRef, internal   // Имя родителя для попап окна, вкладка инфо. При експорте из ECS через скрипт заполняется автоматически, если теги копируются в ручную то требуется в ручную задатать свойство Start Value

HMI tags "2930RS001A01F04"
   "2930RS001A01F04.MSW" : 52809b66-421d-457f-8884-6f7a49d4e247 AT %DB5089.DBX18.0, 500 ms
   "2930RS001A01F04.DefaultText" : TextRef, internal   // Заголовок POPUP окна. При експорте из ECS через скрипт заполняется автоматически, если теги копируются в ручную то требуется в ручную задатать свойство Start Value
   "2930RS001A01F04.BlockInfo" : Array [0..2] of Int AT %DB5089.DBX38.0, 500 ms
   "2930RS001A01F04.StatusWork" : Int AT %DB5089.DBW242, 500 ms
   "2930RS001A01F04.FP_PARAM.DampingTime" : Int AT %DB5089.DBW50, 500 ms
   "2930RS001A01F04.FP_PARAM.Force_Value" : Real AT %DB5089.DBD52, 500 ms
   "2930RS001A01F04.FP_PARAM.Scale_Min" : Real AT %DB5089.DBD56, 500 ms
   "2930RS001A01F04.FP_PARAM.Scale_Max" : Real AT %DB5089.DBD60, 500 ms
   "2930RS001A01F04.FP_PARAM.Gradient" : Real AT %DB5089.DBD64, 500 ms
   "2930RS001A01F04.FP_PARAM.Grad_Pos" : Real AT %DB5089.DBD68, 500 ms
   "2930RS001A01F04.FP_PARAM.Grad_Neg" : Real AT %DB5089.DBD72, 500 ms
   "2930RS001A01F04.FP_PARAM.Grad_X" : Real AT %DB5089.DBD76, 500 ms
   "2930RS001A01F04.FP_PARAM.Gradient_Time_Pre" : Int AT %DB5089.DBW80, 500 ms
   "2930RS001A01F04.FP_PARAM.Gradient_Time_ACC" : Int AT %DB5089.DBW82, 500 ms
   "2930RS001A01F04.FP_PARAM.Alarm_Hyst" : Real AT %DB5089.DBD84, 500 ms
   "2930RS001A01F04.FP_PARAM.AlarmLimit_H3" : Real AT %DB5089.DBD88, 500 ms
   "2930RS001A01F04.FP_PARAM.AlarmLimit_H2" : Real AT %DB5089.DBD92, 500 ms
   "2930RS001A01F04.FP_PARAM.AlarmLimit_H1" : Real AT %DB5089.DBD96, 500 ms
   "2930RS001A01F04.FP_PARAM.AlarmLimit_L1" : Real AT %DB5089.DBD100, 500 ms
   "2930RS001A01F04.FP_PARAM.AlarmLimit_L2" : Real AT %DB5089.DBD104, 500 ms
   "2930RS001A01F04.FP_PARAM.AlarmLimit_L3" : Real AT %DB5089.DBD108, 500 ms
   "2930RS001A01F04.FP_PARAM.AlarmDelay_H3_Pre" : Int AT %DB5089.DBW112, 500 ms
   "2930RS001A01F04.FP_PARAM.AlarmDelay_H3_Acc" : Int AT %DB5089.DBW114, 500 ms
   "2930RS001A01F04.FP_PARAM.AlarmDelay_H2_Pre" : Int AT %DB5089.DBW116, 500 ms
   "2930RS001A01F04.FP_PARAM.AlarmDelay_H2_Acc" : Int AT %DB5089.DBW118, 500 ms
   "2930RS001A01F04.FP_PARAM.AlarmDelay_H1_Pre" : Int AT %DB5089.DBW120, 500 ms
   "2930RS001A01F04.FP_PARAM.AlarmDelay_H1_Acc" : Int AT %DB5089.DBW122, 500 ms
   "2930RS001A01F04.FP_PARAM.AlarmDelay_L1_Pre" : Int AT %DB5089.DBW124, 500 ms
   "2930RS001A01F04.FP_PARAM.AlarmDelay_L1_Acc" : Int AT %DB5089.DBW126, 500 ms
   "2930RS001A01F04.FP_PARAM.AlarmDelay_L2_Pre" : Int AT %DB5089.DBW128, 500 ms
   "2930RS001A01F04.FP_PARAM.AlarmDelay_L2_Acc" : Int AT %DB5089.DBW130, 500 ms
   "2930RS001A01F04.FP_PARAM.AlarmDelay_L3_Pre" : Int AT %DB5089.DBW132, 500 ms
   "2930RS001A01F04.FP_PARAM.AlarmDelay_L3_Acc" : Int AT %DB5089.DBW134, 500 ms
   "2930RS001A01F04.FP_PARAM.OpenLoopDelay_Pre" : Int AT %DB5089.DBW136, 500 ms
   "2930RS001A01F04.FP_PARAM.OpenLoopDelay_Acc" : Int AT %DB5089.DBW138, 500 ms
   "2930RS001A01F04.FP_PARAM.OverRangeDelay_Pre" : Int AT %DB5089.DBW140, 500 ms
   "2930RS001A01F04.FP_PARAM.OverRangeDelay_Acc" : Int AT %DB5089.DBW142, 500 ms
   "2930RS001A01F04.FP_PARAM.AuxLimit_H2_Value" : Real AT %DB5089.DBD144, 500 ms
   "2930RS001A01F04.FP_PARAM.AuxLimit_H1_Value" : Real AT %DB5089.DBD148, 500 ms
   "2930RS001A01F04.FP_PARAM.AuxLimit_L2_Value" : Real AT %DB5089.DBD152, 500 ms
   "2930RS001A01F04.FP_PARAM.AuxLimit_L1_Value" : Real AT %DB5089.DBD156, 500 ms
   "2930RS001A01F04.Unit" : TextRef, internal   // Еденицы измерения При експорте из ECS через скрипт заполняется автоматически, если теги копируются в ручную то требуется задатать свойство Text
   "2930RS001A01F04.Decimals" : TextRef, internal   // Формат отображения При експорте из ECS через скрипт, заполняется автоматически. Если теги копируются в ручную то требуется задатать свойство Text s999999.9
   "2930RS001A01F04.FP_EN.Square" : Bool AT %DB5089.DBX46.0, 500 ms
   "2930RS001A01F04.FP_EN.SquareRoot" : Bool AT %DB5089.DBX46.1, 500 ms
   "2930RS001A01F04.FP_EN.ParentSupress" : Bool AT %DB5089.DBX46.2, 500 ms
   "2930RS001A01F04.FP_EN.ParentSupressUnit" : Bool AT %DB5089.DBX46.3, 500 ms
   "2930RS001A01F04.FP_EN.Force" : Bool AT %DB5089.DBX46.4, 500 ms
   "2930RS001A01F04.FP_EN.Damping" : Bool AT %DB5089.DBX46.5, 500 ms
   "2930RS001A01F04.FP_EN.Gradient_Pos" : Bool AT %DB5089.DBX46.6, 500 ms
   "2930RS001A01F04.FP_EN.Gradient_Neg" : Bool AT %DB5089.DBX46.7, 500 ms
   "2930RS001A01F04.FP_EN.Hysteresis" : Bool AT %DB5089.DBX47.0, 500 ms
   "2930RS001A01F04.FP_EN.Alarm_H3" : Bool AT %DB5089.DBX47.1, 500 ms
   "2930RS001A01F04.FP_EN.Alarm_H2" : Bool AT %DB5089.DBX47.2, 500 ms
   "2930RS001A01F04.FP_EN.Alarm_H1" : Bool AT %DB5089.DBX47.3, 500 ms
   "2930RS001A01F04.FP_EN.Alarm_L1" : Bool AT %DB5089.DBX47.4, 500 ms
   "2930RS001A01F04.FP_EN.Alarm_L2" : Bool AT %DB5089.DBX47.5, 500 ms
   "2930RS001A01F04.FP_EN.Alarm_L3" : Bool AT %DB5089.DBX47.6, 500 ms
   "2930RS001A01F04.FP_EN.AlarmDelay_H3" : Bool AT %DB5089.DBX47.7, 500 ms
   "2930RS001A01F04.FP_EN.AlarmDelay_H2" : Bool AT %DB5089.DBX48.0, 500 ms
   "2930RS001A01F04.FP_EN.AlarmDelay_H1" : Bool AT %DB5089.DBX48.1, 500 ms
   "2930RS001A01F04.FP_EN.AlarmDelay_L1" : Bool AT %DB5089.DBX48.2, 500 ms
   "2930RS001A01F04.FP_EN.AlarmDelay_L2" : Bool AT %DB5089.DBX48.3, 500 ms
   "2930RS001A01F04.FP_EN.AlarmDelay_L3" : Bool AT %DB5089.DBX48.4, 500 ms
   "2930RS001A01F04.FP_EN.ROC_Warn" : Bool AT %DB5089.DBX48.5, 500 ms
   "2930RS001A01F04.FP_EN.U_Range_Warn" : Bool AT %DB5089.DBX48.6, 500 ms
   "2930RS001A01F04.FP_EN.O_Range_Warn" : Bool AT %DB5089.DBX48.7, 500 ms
   "2930RS001A01F04.trend_tag_name" : TextRef, internal   // Еденицы измерения При експорте из ECS через скрипт - заполняется автоматически, если теги копируются в ручную то требуется задатать свойство Text - имя тега для тренда
   "2930RS001A01F04.DQ.AL_H3" : Bool AT %DB5089.DBX16.0, 500 ms
   "2930RS001A01F04.DQ.AL_H2" : Bool AT %DB5089.DBX16.1, 500 ms
   "2930RS001A01F04.DQ.AL_H1" : Bool AT %DB5089.DBX16.2, 500 ms
   "2930RS001A01F04.DQ.AL_L1" : Bool AT %DB5089.DBX16.3, 500 ms
   "2930RS001A01F04.DQ.AL_L2" : Bool AT %DB5089.DBX16.4, 500 ms
   "2930RS001A01F04.DQ.AL_L3" : Bool AT %DB5089.DBX16.5, 500 ms
   "2930RS001A01F04.DQ.SIG_OK" : Bool AT %DB5089.DBX16.6, 500 ms
   "2930RS001A01F04.DQ.LIM_H2" : Bool AT %DB5089.DBX16.7, 500 ms
   "2930RS001A01F04.DQ.LIM_H1" : Bool AT %DB5089.DBX17.0, 500 ms
   "2930RS001A01F04.DQ.LIM_L1" : Bool AT %DB5089.DBX17.1, 500 ms
   "2930RS001A01F04.DQ.LIM_L2" : Bool AT %DB5089.DBX17.2, 500 ms
   "2930RS001A01F04.DQ.GR_P" : Bool AT %DB5089.DBX17.3, 500 ms
   "2930RS001A01F04.DQ.GR_N" : Bool AT %DB5089.DBX17.4, 500 ms
   "2930RS001A01F04.I.IN" : Real AT %DB5089.DBD2, 500 ms
   "2930RS001A01F04.I.SIG_TYPE" : Int AT %DB5089.DBW0, 500 ms
   "2930RS001A01F04.I.FI_BUS" : Byte AT %DB5089.DBB6, 500 ms
   "2930RS001A01F04.DI.U_RANGE" : Bool AT %DB5089.DBX7.0, 500 ms
   "2930RS001A01F04.DI.O_RANGE" : Bool AT %DB5089.DBX7.1, 500 ms
   "2930RS001A01F04.DI.SIG_FAULT" : Bool AT %DB5089.DBX7.2, 500 ms
   "2930RS001A01F04.DI.EnConfig" : Bool AT %DB5089.DBX7.3, 500 ms
   "2930RS001A01F04.DI.AEN" : Bool AT %DB5089.DBX7.4, 500 ms
   "2930RS001A01F04.DI.AL_SUPR" : Bool AT %DB5089.DBX7.5, 500 ms
   "2930RS001A01F04.Q.PV_NORM" : Real AT %DB5089.DBD8, 500 ms
   "2930RS001A01F04.Q.PV_SCAL" : Real AT %DB5089.DBD12, 500 ms
   "2930RS001A01F04.ParentInfo" : TextRef, internal   // Имя родителя для попап окна, вкладка инфо. При експорте из ECS через скрипт заполняется автоматически, если теги копируются в ручную то требуется в ручную задатать свойство Start Value

HMI tags "2930RS001A01F05"
   "2930RS001A01F05.MSW" : 52809b66-421d-457f-8884-6f7a49d4e247 AT %DB5090.DBX18.0, 500 ms
   "2930RS001A01F05.DefaultText" : TextRef, internal   // Заголовок POPUP окна. При експорте из ECS через скрипт заполняется автоматически, если теги копируются в ручную то требуется в ручную задатать свойство Start Value
   "2930RS001A01F05.BlockInfo" : Array [0..2] of Int AT %DB5090.DBX38.0, 500 ms
   "2930RS001A01F05.StatusWork" : Int AT %DB5090.DBW242, 500 ms
   "2930RS001A01F05.FP_PARAM.DampingTime" : Int AT %DB5090.DBW50, 500 ms
   "2930RS001A01F05.FP_PARAM.Force_Value" : Real AT %DB5090.DBD52, 500 ms
   "2930RS001A01F05.FP_PARAM.Scale_Min" : Real AT %DB5090.DBD56, 500 ms
   "2930RS001A01F05.FP_PARAM.Scale_Max" : Real AT %DB5090.DBD60, 500 ms
   "2930RS001A01F05.FP_PARAM.Gradient" : Real AT %DB5090.DBD64, 500 ms
   "2930RS001A01F05.FP_PARAM.Grad_Pos" : Real AT %DB5090.DBD68, 500 ms
   "2930RS001A01F05.FP_PARAM.Grad_Neg" : Real AT %DB5090.DBD72, 500 ms
   "2930RS001A01F05.FP_PARAM.Grad_X" : Real AT %DB5090.DBD76, 500 ms
   "2930RS001A01F05.FP_PARAM.Gradient_Time_Pre" : Int AT %DB5090.DBW80, 500 ms
   "2930RS001A01F05.FP_PARAM.Gradient_Time_ACC" : Int AT %DB5090.DBW82, 500 ms
   "2930RS001A01F05.FP_PARAM.Alarm_Hyst" : Real AT %DB5090.DBD84, 500 ms
   "2930RS001A01F05.FP_PARAM.AlarmLimit_H3" : Real AT %DB5090.DBD88, 500 ms
   "2930RS001A01F05.FP_PARAM.AlarmLimit_H2" : Real AT %DB5090.DBD92, 500 ms
   "2930RS001A01F05.FP_PARAM.AlarmLimit_H1" : Real AT %DB5090.DBD96, 500 ms
   "2930RS001A01F05.FP_PARAM.AlarmLimit_L1" : Real AT %DB5090.DBD100, 500 ms
   "2930RS001A01F05.FP_PARAM.AlarmLimit_L2" : Real AT %DB5090.DBD104, 500 ms
   "2930RS001A01F05.FP_PARAM.AlarmLimit_L3" : Real AT %DB5090.DBD108, 500 ms
   "2930RS001A01F05.FP_PARAM.AlarmDelay_H3_Pre" : Int AT %DB5090.DBW112, 500 ms
   "2930RS001A01F05.FP_PARAM.AlarmDelay_H3_Acc" : Int AT %DB5090.DBW114, 500 ms
   "2930RS001A01F05.FP_PARAM.AlarmDelay_H2_Pre" : Int AT %DB5090.DBW116, 500 ms
   "2930RS001A01F05.FP_PARAM.AlarmDelay_H2_Acc" : Int AT %DB5090.DBW118, 500 ms
   "2930RS001A01F05.FP_PARAM.AlarmDelay_H1_Pre" : Int AT %DB5090.DBW120, 500 ms
   "2930RS001A01F05.FP_PARAM.AlarmDelay_H1_Acc" : Int AT %DB5090.DBW122, 500 ms
   "2930RS001A01F05.FP_PARAM.AlarmDelay_L1_Pre" : Int AT %DB5090.DBW124, 500 ms
   "2930RS001A01F05.FP_PARAM.AlarmDelay_L1_Acc" : Int AT %DB5090.DBW126, 500 ms
   "2930RS001A01F05.FP_PARAM.AlarmDelay_L2_Pre" : Int AT %DB5090.DBW128, 500 ms
   "2930RS001A01F05.FP_PARAM.AlarmDelay_L2_Acc" : Int AT %DB5090.DBW130, 500 ms
   "2930RS001A01F05.FP_PARAM.AlarmDelay_L3_Pre" : Int AT %DB5090.DBW132, 500 ms
   "2930RS001A01F05.FP_PARAM.AlarmDelay_L3_Acc" : Int AT %DB5090.DBW134, 500 ms
   "2930RS001A01F05.FP_PARAM.OpenLoopDelay_Pre" : Int AT %DB5090.DBW136, 500 ms
   "2930RS001A01F05.FP_PARAM.OpenLoopDelay_Acc" : Int AT %DB5090.DBW138, 500 ms
   "2930RS001A01F05.FP_PARAM.OverRangeDelay_Pre" : Int AT %DB5090.DBW140, 500 ms
   "2930RS001A01F05.FP_PARAM.OverRangeDelay_Acc" : Int AT %DB5090.DBW142, 500 ms
   "2930RS001A01F05.FP_PARAM.AuxLimit_H2_Value" : Real AT %DB5090.DBD144, 500 ms
   "2930RS001A01F05.FP_PARAM.AuxLimit_H1_Value" : Real AT %DB5090.DBD148, 500 ms
   "2930RS001A01F05.FP_PARAM.AuxLimit_L2_Value" : Real AT %DB5090.DBD152, 500 ms
   "2930RS001A01F05.FP_PARAM.AuxLimit_L1_Value" : Real AT %DB5090.DBD156, 500 ms
   "2930RS001A01F05.Unit" : TextRef, internal   // Еденицы измерения При експорте из ECS через скрипт заполняется автоматически, если теги копируются в ручную то требуется задатать свойство Text
   "2930RS001A01F05.Decimals" : TextRef, internal   // Формат отображения При експорте из ECS через скрипт, заполняется автоматически. Если теги копируются в ручную то требуется задатать свойство Text s999999.9
   "2930RS001A01F05.FP_EN.Square" : Bool AT %DB5090.DBX46.0, 500 ms
   "2930RS001A01F05.FP_EN.SquareRoot" : Bool AT %DB5090.DBX46.1, 500 ms
   "2930RS001A01F05.FP_EN.ParentSupress" : Bool AT %DB5090.DBX46.2, 500 ms
   "2930RS001A01F05.FP_EN.ParentSupressUnit" : Bool AT %DB5090.DBX46.3, 500 ms
   "2930RS001A01F05.FP_EN.Force" : Bool AT %DB5090.DBX46.4, 500 ms
   "2930RS001A01F05.FP_EN.Damping" : Bool AT %DB5090.DBX46.5, 500 ms
   "2930RS001A01F05.FP_EN.Gradient_Pos" : Bool AT %DB5090.DBX46.6, 500 ms
   "2930RS001A01F05.FP_EN.Gradient_Neg" : Bool AT %DB5090.DBX46.7, 500 ms
   "2930RS001A01F05.FP_EN.Hysteresis" : Bool AT %DB5090.DBX47.0, 500 ms
   "2930RS001A01F05.FP_EN.Alarm_H3" : Bool AT %DB5090.DBX47.1, 500 ms
   "2930RS001A01F05.FP_EN.Alarm_H2" : Bool AT %DB5090.DBX47.2, 500 ms
   "2930RS001A01F05.FP_EN.Alarm_H1" : Bool AT %DB5090.DBX47.3, 500 ms
   "2930RS001A01F05.FP_EN.Alarm_L1" : Bool AT %DB5090.DBX47.4, 500 ms
   "2930RS001A01F05.FP_EN.Alarm_L2" : Bool AT %DB5090.DBX47.5, 500 ms
   "2930RS001A01F05.FP_EN.Alarm_L3" : Bool AT %DB5090.DBX47.6, 500 ms
   "2930RS001A01F05.FP_EN.AlarmDelay_H3" : Bool AT %DB5090.DBX47.7, 500 ms
   "2930RS001A01F05.FP_EN.AlarmDelay_H2" : Bool AT %DB5090.DBX48.0, 500 ms
   "2930RS001A01F05.FP_EN.AlarmDelay_H1" : Bool AT %DB5090.DBX48.1, 500 ms
   "2930RS001A01F05.FP_EN.AlarmDelay_L1" : Bool AT %DB5090.DBX48.2, 500 ms
   "2930RS001A01F05.FP_EN.AlarmDelay_L2" : Bool AT %DB5090.DBX48.3, 500 ms
   "2930RS001A01F05.FP_EN.AlarmDelay_L3" : Bool AT %DB5090.DBX48.4, 500 ms
   "2930RS001A01F05.FP_EN.ROC_Warn" : Bool AT %DB5090.DBX48.5, 500 ms
   "2930RS001A01F05.FP_EN.U_Range_Warn" : Bool AT %DB5090.DBX48.6, 500 ms
   "2930RS001A01F05.FP_EN.O_Range_Warn" : Bool AT %DB5090.DBX48.7, 500 ms
   "2930RS001A01F05.trend_tag_name" : TextRef, internal   // Еденицы измерения При експорте из ECS через скрипт - заполняется автоматически, если теги копируются в ручную то требуется задатать свойство Text - имя тега для тренда
   "2930RS001A01F05.DQ.AL_H3" : Bool AT %DB5090.DBX16.0, 500 ms
   "2930RS001A01F05.DQ.AL_H2" : Bool AT %DB5090.DBX16.1, 500 ms
   "2930RS001A01F05.DQ.AL_H1" : Bool AT %DB5090.DBX16.2, 500 ms
   "2930RS001A01F05.DQ.AL_L1" : Bool AT %DB5090.DBX16.3, 500 ms
   "2930RS001A01F05.DQ.AL_L2" : Bool AT %DB5090.DBX16.4, 500 ms
   "2930RS001A01F05.DQ.AL_L3" : Bool AT %DB5090.DBX16.5, 500 ms
   "2930RS001A01F05.DQ.SIG_OK" : Bool AT %DB5090.DBX16.6, 500 ms
   "2930RS001A01F05.DQ.LIM_H2" : Bool AT %DB5090.DBX16.7, 500 ms
   "2930RS001A01F05.DQ.LIM_H1" : Bool AT %DB5090.DBX17.0, 500 ms
   "2930RS001A01F05.DQ.LIM_L1" : Bool AT %DB5090.DBX17.1, 500 ms
   "2930RS001A01F05.DQ.LIM_L2" : Bool AT %DB5090.DBX17.2, 500 ms
   "2930RS001A01F05.DQ.GR_P" : Bool AT %DB5090.DBX17.3, 500 ms
   "2930RS001A01F05.DQ.GR_N" : Bool AT %DB5090.DBX17.4, 500 ms
   "2930RS001A01F05.I.IN" : Real AT %DB5090.DBD2, 500 ms
   "2930RS001A01F05.I.SIG_TYPE" : Int AT %DB5090.DBW0, 500 ms
   "2930RS001A01F05.I.FI_BUS" : Byte AT %DB5090.DBB6, 500 ms
   "2930RS001A01F05.DI.U_RANGE" : Bool AT %DB5090.DBX7.0, 500 ms
   "2930RS001A01F05.DI.O_RANGE" : Bool AT %DB5090.DBX7.1, 500 ms
   "2930RS001A01F05.DI.SIG_FAULT" : Bool AT %DB5090.DBX7.2, 500 ms
   "2930RS001A01F05.DI.EnConfig" : Bool AT %DB5090.DBX7.3, 500 ms
   "2930RS001A01F05.DI.AEN" : Bool AT %DB5090.DBX7.4, 500 ms
   "2930RS001A01F05.DI.AL_SUPR" : Bool AT %DB5090.DBX7.5, 500 ms
   "2930RS001A01F05.Q.PV_NORM" : Real AT %DB5090.DBD8, 500 ms
   "2930RS001A01F05.Q.PV_SCAL" : Real AT %DB5090.DBD12, 500 ms
   "2930RS001A01F05.ParentInfo" : TextRef, internal   // Имя родителя для попап окна, вкладка инфо. При експорте из ECS через скрипт заполняется автоматически, если теги копируются в ручную то требуется в ручную задатать свойство Start Value

HMI tags "2930RS001A01F06"
   "2930RS001A01F06.MSW" : 52809b66-421d-457f-8884-6f7a49d4e247 AT %DB5091.DBX18.0, 500 ms
   "2930RS001A01F06.DefaultText" : TextRef, internal   // Заголовок POPUP окна. При експорте из ECS через скрипт заполняется автоматически, если теги копируются в ручную то требуется в ручную задатать свойство Start Value
   "2930RS001A01F06.BlockInfo" : Array [0..2] of Int AT %DB5091.DBX38.0, 500 ms
   "2930RS001A01F06.StatusWork" : Int AT %DB5091.DBW242, 500 ms
   "2930RS001A01F06.FP_PARAM.DampingTime" : Int AT %DB5091.DBW50, 500 ms
   "2930RS001A01F06.FP_PARAM.Force_Value" : Real AT %DB5091.DBD52, 500 ms
   "2930RS001A01F06.FP_PARAM.Scale_Min" : Real AT %DB5091.DBD56, 500 ms
   "2930RS001A01F06.FP_PARAM.Scale_Max" : Real AT %DB5091.DBD60, 500 ms
   "2930RS001A01F06.FP_PARAM.Gradient" : Real AT %DB5091.DBD64, 500 ms
   "2930RS001A01F06.FP_PARAM.Grad_Pos" : Real AT %DB5091.DBD68, 500 ms
   "2930RS001A01F06.FP_PARAM.Grad_Neg" : Real AT %DB5091.DBD72, 500 ms
   "2930RS001A01F06.FP_PARAM.Grad_X" : Real AT %DB5091.DBD76, 500 ms
   "2930RS001A01F06.FP_PARAM.Gradient_Time_Pre" : Int AT %DB5091.DBW80, 500 ms
   "2930RS001A01F06.FP_PARAM.Gradient_Time_ACC" : Int AT %DB5091.DBW82, 500 ms
   "2930RS001A01F06.FP_PARAM.Alarm_Hyst" : Real AT %DB5091.DBD84, 500 ms
   "2930RS001A01F06.FP_PARAM.AlarmLimit_H3" : Real AT %DB5091.DBD88, 500 ms
   "2930RS001A01F06.FP_PARAM.AlarmLimit_H2" : Real AT %DB5091.DBD92, 500 ms
   "2930RS001A01F06.FP_PARAM.AlarmLimit_H1" : Real AT %DB5091.DBD96, 500 ms
   "2930RS001A01F06.FP_PARAM.AlarmLimit_L1" : Real AT %DB5091.DBD100, 500 ms
   "2930RS001A01F06.FP_PARAM.AlarmLimit_L2" : Real AT %DB5091.DBD104, 500 ms
   "2930RS001A01F06.FP_PARAM.AlarmLimit_L3" : Real AT %DB5091.DBD108, 500 ms
   "2930RS001A01F06.FP_PARAM.AlarmDelay_H3_Pre" : Int AT %DB5091.DBW112, 500 ms
   "2930RS001A01F06.FP_PARAM.AlarmDelay_H3_Acc" : Int AT %DB5091.DBW114, 500 ms
   "2930RS001A01F06.FP_PARAM.AlarmDelay_H2_Pre" : Int AT %DB5091.DBW116, 500 ms
   "2930RS001A01F06.FP_PARAM.AlarmDelay_H2_Acc" : Int AT %DB5091.DBW118, 500 ms
   "2930RS001A01F06.FP_PARAM.AlarmDelay_H1_Pre" : Int AT %DB5091.DBW120, 500 ms
   "2930RS001A01F06.FP_PARAM.AlarmDelay_H1_Acc" : Int AT %DB5091.DBW122, 500 ms
   "2930RS001A01F06.FP_PARAM.AlarmDelay_L1_Pre" : Int AT %DB5091.DBW124, 500 ms
   "2930RS001A01F06.FP_PARAM.AlarmDelay_L1_Acc" : Int AT %DB5091.DBW126, 500 ms
   "2930RS001A01F06.FP_PARAM.AlarmDelay_L2_Pre" : Int AT %DB5091.DBW128, 500 ms
   "2930RS001A01F06.FP_PARAM.AlarmDelay_L2_Acc" : Int AT %DB5091.DBW130, 500 ms
   "2930RS001A01F06.FP_PARAM.AlarmDelay_L3_Pre" : Int AT %DB5091.DBW132, 500 ms
   "2930RS001A01F06.FP_PARAM.AlarmDelay_L3_Acc" : Int AT %DB5091.DBW134, 500 ms
   "2930RS001A01F06.FP_PARAM.OpenLoopDelay_Pre" : Int AT %DB5091.DBW136, 500 ms
   "2930RS001A01F06.FP_PARAM.OpenLoopDelay_Acc" : Int AT %DB5091.DBW138, 500 ms
   "2930RS001A01F06.FP_PARAM.OverRangeDelay_Pre" : Int AT %DB5091.DBW140, 500 ms
   "2930RS001A01F06.FP_PARAM.OverRangeDelay_Acc" : Int AT %DB5091.DBW142, 500 ms
   "2930RS001A01F06.FP_PARAM.AuxLimit_H2_Value" : Real AT %DB5091.DBD144, 500 ms
   "2930RS001A01F06.FP_PARAM.AuxLimit_H1_Value" : Real AT %DB5091.DBD148, 500 ms
   "2930RS001A01F06.FP_PARAM.AuxLimit_L2_Value" : Real AT %DB5091.DBD152, 500 ms
   "2930RS001A01F06.FP_PARAM.AuxLimit_L1_Value" : Real AT %DB5091.DBD156, 500 ms
   "2930RS001A01F06.Unit" : TextRef, internal   // Еденицы измерения При експорте из ECS через скрипт заполняется автоматически, если теги копируются в ручную то требуется задатать свойство Text
   "2930RS001A01F06.Decimals" : TextRef, internal   // Формат отображения При експорте из ECS через скрипт, заполняется автоматически. Если теги копируются в ручную то требуется задатать свойство Text s999999.9
   "2930RS001A01F06.FP_EN.Square" : Bool AT %DB5091.DBX46.0, 500 ms
   "2930RS001A01F06.FP_EN.SquareRoot" : Bool AT %DB5091.DBX46.1, 500 ms
   "2930RS001A01F06.FP_EN.ParentSupress" : Bool AT %DB5091.DBX46.2, 500 ms
   "2930RS001A01F06.FP_EN.ParentSupressUnit" : Bool AT %DB5091.DBX46.3, 500 ms
   "2930RS001A01F06.FP_EN.Force" : Bool AT %DB5091.DBX46.4, 500 ms
   "2930RS001A01F06.FP_EN.Damping" : Bool AT %DB5091.DBX46.5, 500 ms
   "2930RS001A01F06.FP_EN.Gradient_Pos" : Bool AT %DB5091.DBX46.6, 500 ms
   "2930RS001A01F06.FP_EN.Gradient_Neg" : Bool AT %DB5091.DBX46.7, 500 ms
   "2930RS001A01F06.FP_EN.Hysteresis" : Bool AT %DB5091.DBX47.0, 500 ms
   "2930RS001A01F06.FP_EN.Alarm_H3" : Bool AT %DB5091.DBX47.1, 500 ms
   "2930RS001A01F06.FP_EN.Alarm_H2" : Bool AT %DB5091.DBX47.2, 500 ms
   "2930RS001A01F06.FP_EN.Alarm_H1" : Bool AT %DB5091.DBX47.3, 500 ms
   "2930RS001A01F06.FP_EN.Alarm_L1" : Bool AT %DB5091.DBX47.4, 500 ms
   "2930RS001A01F06.FP_EN.Alarm_L2" : Bool AT %DB5091.DBX47.5, 500 ms
   "2930RS001A01F06.FP_EN.Alarm_L3" : Bool AT %DB5091.DBX47.6, 500 ms
   "2930RS001A01F06.FP_EN.AlarmDelay_H3" : Bool AT %DB5091.DBX47.7, 500 ms
   "2930RS001A01F06.FP_EN.AlarmDelay_H2" : Bool AT %DB5091.DBX48.0, 500 ms
   "2930RS001A01F06.FP_EN.AlarmDelay_H1" : Bool AT %DB5091.DBX48.1, 500 ms
   "2930RS001A01F06.FP_EN.AlarmDelay_L1" : Bool AT %DB5091.DBX48.2, 500 ms
   "2930RS001A01F06.FP_EN.AlarmDelay_L2" : Bool AT %DB5091.DBX48.3, 500 ms
   "2930RS001A01F06.FP_EN.AlarmDelay_L3" : Bool AT %DB5091.DBX48.4, 500 ms
   "2930RS001A01F06.FP_EN.ROC_Warn" : Bool AT %DB5091.DBX48.5, 500 ms
   "2930RS001A01F06.FP_EN.U_Range_Warn" : Bool AT %DB5091.DBX48.6, 500 ms
   "2930RS001A01F06.FP_EN.O_Range_Warn" : Bool AT %DB5091.DBX48.7, 500 ms
   "2930RS001A01F06.trend_tag_name" : TextRef, internal   // Еденицы измерения При експорте из ECS через скрипт - заполняется автоматически, если теги копируются в ручную то требуется задатать свойство Text - имя тега для тренда
   "2930RS001A01F06.DQ.AL_H3" : Bool AT %DB5091.DBX16.0, 500 ms
   "2930RS001A01F06.DQ.AL_H2" : Bool AT %DB5091.DBX16.1, 500 ms
   "2930RS001A01F06.DQ.AL_H1" : Bool AT %DB5091.DBX16.2, 500 ms
   "2930RS001A01F06.DQ.AL_L1" : Bool AT %DB5091.DBX16.3, 500 ms
   "2930RS001A01F06.DQ.AL_L2" : Bool AT %DB5091.DBX16.4, 500 ms
   "2930RS001A01F06.DQ.AL_L3" : Bool AT %DB5091.DBX16.5, 500 ms
   "2930RS001A01F06.DQ.SIG_OK" : Bool AT %DB5091.DBX16.6, 500 ms
   "2930RS001A01F06.DQ.LIM_H2" : Bool AT %DB5091.DBX16.7, 500 ms
   "2930RS001A01F06.DQ.LIM_H1" : Bool AT %DB5091.DBX17.0, 500 ms
   "2930RS001A01F06.DQ.LIM_L1" : Bool AT %DB5091.DBX17.1, 500 ms
   "2930RS001A01F06.DQ.LIM_L2" : Bool AT %DB5091.DBX17.2, 500 ms
   "2930RS001A01F06.DQ.GR_P" : Bool AT %DB5091.DBX17.3, 500 ms
   "2930RS001A01F06.DQ.GR_N" : Bool AT %DB5091.DBX17.4, 500 ms
   "2930RS001A01F06.I.IN" : Real AT %DB5091.DBD2, 500 ms
   "2930RS001A01F06.I.SIG_TYPE" : Int AT %DB5091.DBW0, 500 ms
   "2930RS001A01F06.I.FI_BUS" : Byte AT %DB5091.DBB6, 500 ms
   "2930RS001A01F06.DI.U_RANGE" : Bool AT %DB5091.DBX7.0, 500 ms
   "2930RS001A01F06.DI.O_RANGE" : Bool AT %DB5091.DBX7.1, 500 ms
   "2930RS001A01F06.DI.SIG_FAULT" : Bool AT %DB5091.DBX7.2, 500 ms
   "2930RS001A01F06.DI.EnConfig" : Bool AT %DB5091.DBX7.3, 500 ms
   "2930RS001A01F06.DI.AEN" : Bool AT %DB5091.DBX7.4, 500 ms
   "2930RS001A01F06.DI.AL_SUPR" : Bool AT %DB5091.DBX7.5, 500 ms
   "2930RS001A01F06.Q.PV_NORM" : Real AT %DB5091.DBD8, 500 ms
   "2930RS001A01F06.Q.PV_SCAL" : Real AT %DB5091.DBD12, 500 ms
   "2930RS001A01F06.ParentInfo" : TextRef, internal   // Имя родителя для попап окна, вкладка инфо. При експорте из ECS через скрипт заполняется автоматически, если теги копируются в ручную то требуется в ручную задатать свойство Start Value

HMI tags "2930RS001A01F07"
   "2930RS001A01F07.MSW" : 52809b66-421d-457f-8884-6f7a49d4e247 AT %DB5092.DBX18.0, 500 ms
   "2930RS001A01F07.DefaultText" : TextRef, internal   // Заголовок POPUP окна. При експорте из ECS через скрипт заполняется автоматически, если теги копируются в ручную то требуется в ручную задатать свойство Start Value
   "2930RS001A01F07.BlockInfo" : Array [0..2] of Int AT %DB5092.DBX38.0, 500 ms
   "2930RS001A01F07.StatusWork" : Int AT %DB5092.DBW242, 500 ms
   "2930RS001A01F07.FP_PARAM.DampingTime" : Int AT %DB5092.DBW50, 500 ms
   "2930RS001A01F07.FP_PARAM.Force_Value" : Real AT %DB5092.DBD52, 500 ms
   "2930RS001A01F07.FP_PARAM.Scale_Min" : Real AT %DB5092.DBD56, 500 ms
   "2930RS001A01F07.FP_PARAM.Scale_Max" : Real AT %DB5092.DBD60, 500 ms
   "2930RS001A01F07.FP_PARAM.Gradient" : Real AT %DB5092.DBD64, 500 ms
   "2930RS001A01F07.FP_PARAM.Grad_Pos" : Real AT %DB5092.DBD68, 500 ms
   "2930RS001A01F07.FP_PARAM.Grad_Neg" : Real AT %DB5092.DBD72, 500 ms
   "2930RS001A01F07.FP_PARAM.Grad_X" : Real AT %DB5092.DBD76, 500 ms
   "2930RS001A01F07.FP_PARAM.Gradient_Time_Pre" : Int AT %DB5092.DBW80, 500 ms
   "2930RS001A01F07.FP_PARAM.Gradient_Time_ACC" : Int AT %DB5092.DBW82, 500 ms
   "2930RS001A01F07.FP_PARAM.Alarm_Hyst" : Real AT %DB5092.DBD84, 500 ms
   "2930RS001A01F07.FP_PARAM.AlarmLimit_H3" : Real AT %DB5092.DBD88, 500 ms
   "2930RS001A01F07.FP_PARAM.AlarmLimit_H2" : Real AT %DB5092.DBD92, 500 ms
   "2930RS001A01F07.FP_PARAM.AlarmLimit_H1" : Real AT %DB5092.DBD96, 500 ms
   "2930RS001A01F07.FP_PARAM.AlarmLimit_L1" : Real AT %DB5092.DBD100, 500 ms
   "2930RS001A01F07.FP_PARAM.AlarmLimit_L2" : Real AT %DB5092.DBD104, 500 ms
   "2930RS001A01F07.FP_PARAM.AlarmLimit_L3" : Real AT %DB5092.DBD108, 500 ms
   "2930RS001A01F07.FP_PARAM.AlarmDelay_H3_Pre" : Int AT %DB5092.DBW112, 500 ms
   "2930RS001A01F07.FP_PARAM.AlarmDelay_H3_Acc" : Int AT %DB5092.DBW114, 500 ms
   "2930RS001A01F07.FP_PARAM.AlarmDelay_H2_Pre" : Int AT %DB5092.DBW116, 500 ms
   "2930RS001A01F07.FP_PARAM.AlarmDelay_H2_Acc" : Int AT %DB5092.DBW118, 500 ms
   "2930RS001A01F07.FP_PARAM.AlarmDelay_H1_Pre" : Int AT %DB5092.DBW120, 500 ms
   "2930RS001A01F07.FP_PARAM.AlarmDelay_H1_Acc" : Int AT %DB5092.DBW122, 500 ms
   "2930RS001A01F07.FP_PARAM.AlarmDelay_L1_Pre" : Int AT %DB5092.DBW124, 500 ms
   "2930RS001A01F07.FP_PARAM.AlarmDelay_L1_Acc" : Int AT %DB5092.DBW126, 500 ms
   "2930RS001A01F07.FP_PARAM.AlarmDelay_L2_Pre" : Int AT %DB5092.DBW128, 500 ms
   "2930RS001A01F07.FP_PARAM.AlarmDelay_L2_Acc" : Int AT %DB5092.DBW130, 500 ms
   "2930RS001A01F07.FP_PARAM.AlarmDelay_L3_Pre" : Int AT %DB5092.DBW132, 500 ms
   "2930RS001A01F07.FP_PARAM.AlarmDelay_L3_Acc" : Int AT %DB5092.DBW134, 500 ms
   "2930RS001A01F07.FP_PARAM.OpenLoopDelay_Pre" : Int AT %DB5092.DBW136, 500 ms
   "2930RS001A01F07.FP_PARAM.OpenLoopDelay_Acc" : Int AT %DB5092.DBW138, 500 ms
   "2930RS001A01F07.FP_PARAM.OverRangeDelay_Pre" : Int AT %DB5092.DBW140, 500 ms
   "2930RS001A01F07.FP_PARAM.OverRangeDelay_Acc" : Int AT %DB5092.DBW142, 500 ms
   "2930RS001A01F07.FP_PARAM.AuxLimit_H2_Value" : Real AT %DB5092.DBD144, 500 ms
   "2930RS001A01F07.FP_PARAM.AuxLimit_H1_Value" : Real AT %DB5092.DBD148, 500 ms
   "2930RS001A01F07.FP_PARAM.AuxLimit_L2_Value" : Real AT %DB5092.DBD152, 500 ms
   "2930RS001A01F07.FP_PARAM.AuxLimit_L1_Value" : Real AT %DB5092.DBD156, 500 ms
   "2930RS001A01F07.Unit" : TextRef, internal   // Еденицы измерения При експорте из ECS через скрипт заполняется автоматически, если теги копируются в ручную то требуется задатать свойство Text
   "2930RS001A01F07.Decimals" : TextRef, internal   // Формат отображения При експорте из ECS через скрипт, заполняется автоматически. Если теги копируются в ручную то требуется задатать свойство Text s999999.9
   "2930RS001A01F07.FP_EN.Square" : Bool AT %DB5092.DBX46.0, 500 ms
   "2930RS001A01F07.FP_EN.SquareRoot" : Bool AT %DB5092.DBX46.1, 500 ms
   "2930RS001A01F07.FP_EN.ParentSupress" : Bool AT %DB5092.DBX46.2, 500 ms
   "2930RS001A01F07.FP_EN.ParentSupressUnit" : Bool AT %DB5092.DBX46.3, 500 ms
   "2930RS001A01F07.FP_EN.Force" : Bool AT %DB5092.DBX46.4, 500 ms
   "2930RS001A01F07.FP_EN.Damping" : Bool AT %DB5092.DBX46.5, 500 ms
   "2930RS001A01F07.FP_EN.Gradient_Pos" : Bool AT %DB5092.DBX46.6, 500 ms
   "2930RS001A01F07.FP_EN.Gradient_Neg" : Bool AT %DB5092.DBX46.7, 500 ms
   "2930RS001A01F07.FP_EN.Hysteresis" : Bool AT %DB5092.DBX47.0, 500 ms
   "2930RS001A01F07.FP_EN.Alarm_H3" : Bool AT %DB5092.DBX47.1, 500 ms
   "2930RS001A01F07.FP_EN.Alarm_H2" : Bool AT %DB5092.DBX47.2, 500 ms
   "2930RS001A01F07.FP_EN.Alarm_H1" : Bool AT %DB5092.DBX47.3, 500 ms
   "2930RS001A01F07.FP_EN.Alarm_L1" : Bool AT %DB5092.DBX47.4, 500 ms
   "2930RS001A01F07.FP_EN.Alarm_L2" : Bool AT %DB5092.DBX47.5, 500 ms
   "2930RS001A01F07.FP_EN.Alarm_L3" : Bool AT %DB5092.DBX47.6, 500 ms
   "2930RS001A01F07.FP_EN.AlarmDelay_H3" : Bool AT %DB5092.DBX47.7, 500 ms
   "2930RS001A01F07.FP_EN.AlarmDelay_H2" : Bool AT %DB5092.DBX48.0, 500 ms
   "2930RS001A01F07.FP_EN.AlarmDelay_H1" : Bool AT %DB5092.DBX48.1, 500 ms
   "2930RS001A01F07.FP_EN.AlarmDelay_L1" : Bool AT %DB5092.DBX48.2, 500 ms
   "2930RS001A01F07.FP_EN.AlarmDelay_L2" : Bool AT %DB5092.DBX48.3, 500 ms
   "2930RS001A01F07.FP_EN.AlarmDelay_L3" : Bool AT %DB5092.DBX48.4, 500 ms
   "2930RS001A01F07.FP_EN.ROC_Warn" : Bool AT %DB5092.DBX48.5, 500 ms
   "2930RS001A01F07.FP_EN.U_Range_Warn" : Bool AT %DB5092.DBX48.6, 500 ms
   "2930RS001A01F07.FP_EN.O_Range_Warn" : Bool AT %DB5092.DBX48.7, 500 ms
   "2930RS001A01F07.trend_tag_name" : TextRef, internal   // Еденицы измерения При експорте из ECS через скрипт - заполняется автоматически, если теги копируются в ручную то требуется задатать свойство Text - имя тега для тренда
   "2930RS001A01F07.DQ.AL_H3" : Bool AT %DB5092.DBX16.0, 500 ms
   "2930RS001A01F07.DQ.AL_H2" : Bool AT %DB5092.DBX16.1, 500 ms
   "2930RS001A01F07.DQ.AL_H1" : Bool AT %DB5092.DBX16.2, 500 ms
   "2930RS001A01F07.DQ.AL_L1" : Bool AT %DB5092.DBX16.3, 500 ms
   "2930RS001A01F07.DQ.AL_L2" : Bool AT %DB5092.DBX16.4, 500 ms
   "2930RS001A01F07.DQ.AL_L3" : Bool AT %DB5092.DBX16.5, 500 ms
   "2930RS001A01F07.DQ.SIG_OK" : Bool AT %DB5092.DBX16.6, 500 ms
   "2930RS001A01F07.DQ.LIM_H2" : Bool AT %DB5092.DBX16.7, 500 ms
   "2930RS001A01F07.DQ.LIM_H1" : Bool AT %DB5092.DBX17.0, 500 ms
   "2930RS001A01F07.DQ.LIM_L1" : Bool AT %DB5092.DBX17.1, 500 ms
   "2930RS001A01F07.DQ.LIM_L2" : Bool AT %DB5092.DBX17.2, 500 ms
   "2930RS001A01F07.DQ.GR_P" : Bool AT %DB5092.DBX17.3, 500 ms
   "2930RS001A01F07.DQ.GR_N" : Bool AT %DB5092.DBX17.4, 500 ms
   "2930RS001A01F07.I.IN" : Real AT %DB5092.DBD2, 500 ms
   "2930RS001A01F07.I.SIG_TYPE" : Int AT %DB5092.DBW0, 500 ms
   "2930RS001A01F07.I.FI_BUS" : Byte AT %DB5092.DBB6, 500 ms
   "2930RS001A01F07.DI.U_RANGE" : Bool AT %DB5092.DBX7.0, 500 ms
   "2930RS001A01F07.DI.O_RANGE" : Bool AT %DB5092.DBX7.1, 500 ms
   "2930RS001A01F07.DI.SIG_FAULT" : Bool AT %DB5092.DBX7.2, 500 ms
   "2930RS001A01F07.DI.EnConfig" : Bool AT %DB5092.DBX7.3, 500 ms
   "2930RS001A01F07.DI.AEN" : Bool AT %DB5092.DBX7.4, 500 ms
   "2930RS001A01F07.DI.AL_SUPR" : Bool AT %DB5092.DBX7.5, 500 ms
   "2930RS001A01F07.Q.PV_NORM" : Real AT %DB5092.DBD8, 500 ms
   "2930RS001A01F07.Q.PV_SCAL" : Real AT %DB5092.DBD12, 500 ms
   "2930RS001A01F07.ParentInfo" : TextRef, internal   // Имя родителя для попап окна, вкладка инфо. При експорте из ECS через скрипт заполняется автоматически, если теги копируются в ручную то требуется в ручную задатать свойство Start Value

